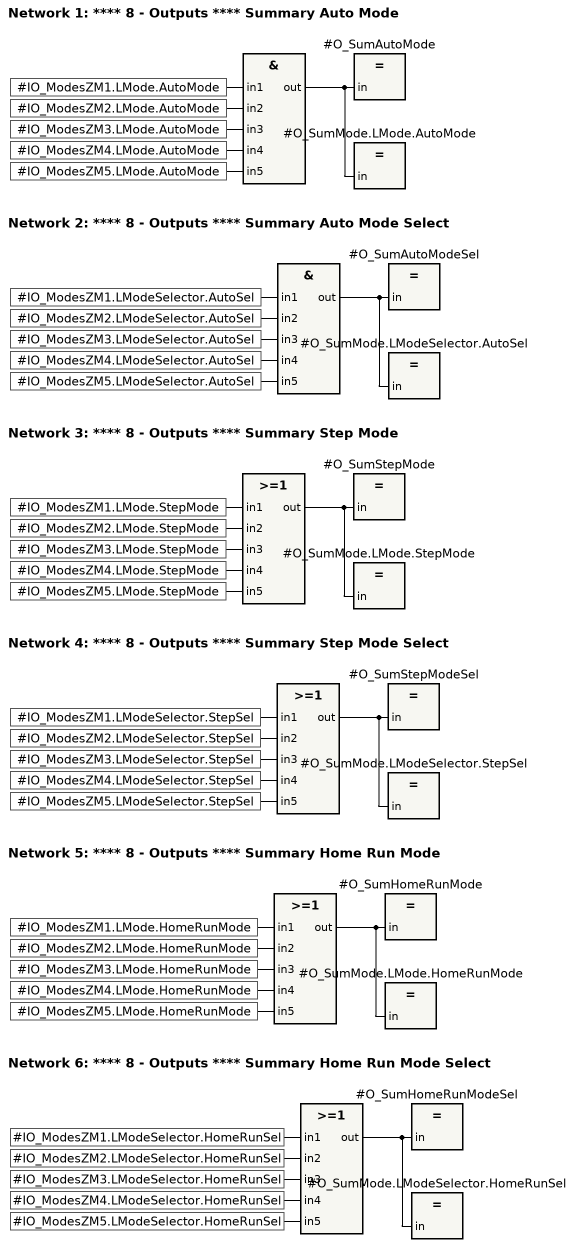
   #O_SumAutoMode := #IO_ModesZM1.LMode.AutoMode AND #IO_ModesZM2.LMode.AutoMode AND #IO_ModesZM3.LMode.AutoMode AND #IO_ModesZM4.LMode.AutoMode AND #IO_ModesZM5.LMode.AutoMode;
   #O_SumMode.LMode.AutoMode := #O_SumAutoMode;
END_REGION

REGION Network 2: **** 8 - Outputs **** Summary Auto Mode Select
   #O_SumAutoModeSel := #IO_ModesZM1.LModeSelector.AutoSel AND #IO_ModesZM2.LModeSelector.AutoSel AND #IO_ModesZM3.LModeSelector.AutoSel AND #IO_ModesZM4.LModeSelector.AutoSel AND #IO_ModesZM5.LModeSelector.AutoSel;
   #O_SumMode.LModeSelector.AutoSel := #O_SumAutoModeSel;
END_REGION

REGION Network 3: **** 8 - Outputs **** Summary Step Mode
   #O_SumStepMode := #IO_ModesZM1.LMode.StepMode OR #IO_ModesZM2.LMode.StepMode OR #IO_ModesZM3.LMode.StepMode OR #IO_ModesZM4.LMode.StepMode OR #IO_ModesZM5.LMode.StepMode;
   #O_SumMode.LMode.StepMode := #O_SumStepMode;
END_REGION

REGION Network 4: **** 8 - Outputs **** Summary Step Mode Select
   #O_SumStepModeSel := #IO_ModesZM1.LModeSelector.StepSel OR #IO_ModesZM2.LModeSelector.StepSel OR #IO_ModesZM3.LModeSelector.StepSel OR #IO_ModesZM4.LModeSelector.StepSel OR #IO_ModesZM5.LModeSelector.StepSel;
   #O_SumMode.LModeSelector.StepSel := #O_SumStepModeSel;
END_REGION

REGION Network 5: **** 8 - Outputs **** Summary Home Run Mode
   #O_SumHomeRunMode := #IO_ModesZM1.LMode.HomeRunMode OR #IO_ModesZM2.LMode.HomeRunMode OR #IO_ModesZM3.LMode.HomeRunMode OR #IO_ModesZM4.LMode.HomeRunMode OR #IO_ModesZM5.LMode.HomeRunMode;
   #O_SumMode.LMode.HomeRunMode := #O_SumHomeRunMode;
END_REGION

REGION Network 6: **** 8 - Outputs **** Summary Home Run Mode Select
   #O_SumHomeRunModeSel := #IO_ModesZM1.LModeSelector.HomeRunSel OR #IO_ModesZM2.LModeSelector.HomeRunSel OR #IO_ModesZM3.LModeSelector.HomeRunSel OR #IO_ModesZM4.LModeSelector.HomeRunSel OR #IO_ModesZM5.LModeSelector.HomeRunSel;
   #O_SumMode.LModeSelector.HomeRunSel := #O_SumHomeRunModeSel;
END_REGION

REGION Network 7: **** 8 - Outputs **** Summary Manual Mode
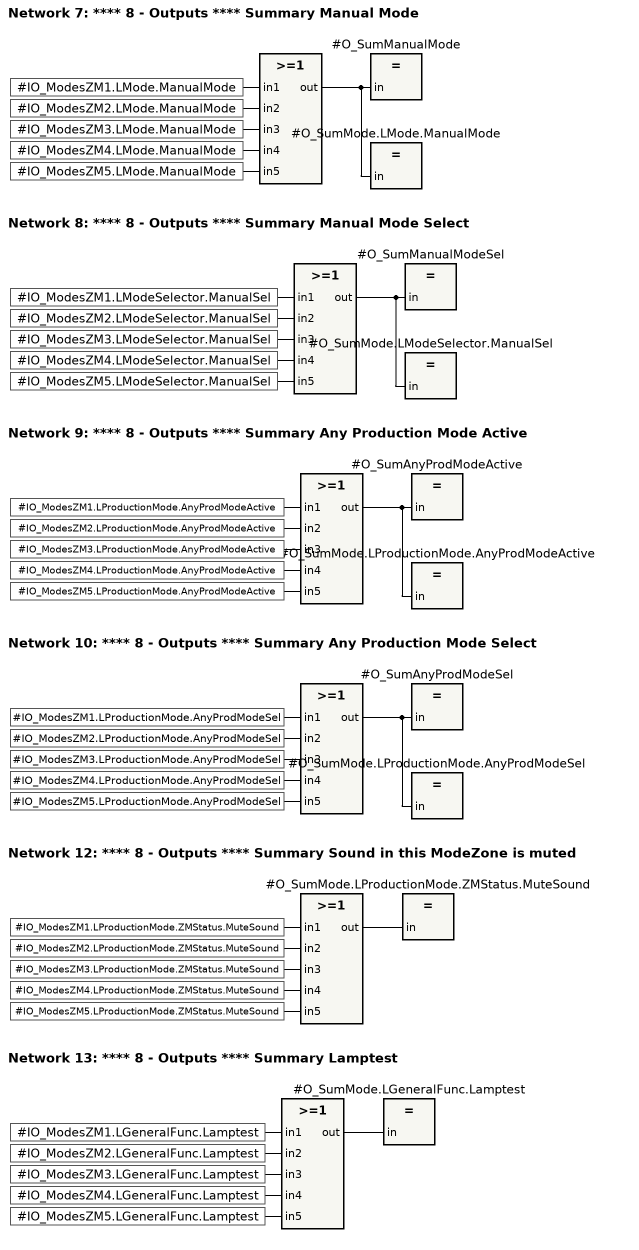
   #O_SumManualMode := #IO_ModesZM1.LMode.ManualMode OR #IO_ModesZM2.LMode.ManualMode OR #IO_ModesZM3.LMode.ManualMode OR #IO_ModesZM4.LMode.ManualMode OR #IO_ModesZM5.LMode.ManualMode;
   #O_SumMode.LMode.ManualMode := #O_SumManualMode;
END_REGION

REGION Network 8: **** 8 - Outputs **** Summary Manual Mode Select
   #O_SumManualModeSel := #IO_ModesZM1.LModeSelector.ManualSel OR #IO_ModesZM2.LModeSelector.ManualSel OR #IO_ModesZM3.LModeSelector.ManualSel OR #IO_ModesZM4.LModeSelector.ManualSel OR #IO_ModesZM5.LModeSelector.ManualSel;
   #O_SumMode.LModeSelector.ManualSel := #O_SumManualModeSel;
END_REGION

REGION Network 9: **** 8 - Outputs **** Summary Any Production Mode Active
   #O_SumAnyProdModeActive := #IO_ModesZM1.LProductionMode.AnyProdModeActive OR #IO_ModesZM2.LProductionMode.AnyProdModeActive OR #IO_ModesZM3.LProductionMode.AnyProdModeActive OR #IO_ModesZM4.LProductionMode.AnyProdModeActive OR #IO_ModesZM5.LProductionMode.AnyProdModeActive;
   #O_SumMode.LProductionMode.AnyProdModeActive := #O_SumAnyProdModeActive;
END_REGION

REGION Network 10: **** 8 - Outputs **** Summary Any Production Mode Select
   #O_SumAnyProdModeSel := #IO_ModesZM1.LProductionMode.AnyProdModeSel OR #IO_ModesZM2.LProductionMode.AnyProdModeSel OR #IO_ModesZM3.LProductionMode.AnyProdModeSel OR #IO_ModesZM4.LProductionMode.AnyProdModeSel OR #IO_ModesZM5.LProductionMode.AnyProdModeSel;
   #O_SumMode.LProductionMode.AnyProdModeSel := #O_SumAnyProdModeSel;
END_REGION

REGION Network 11: **** --------------------- Extra --------------------- ****
END_REGION

REGION Network 12: **** 8 - Outputs **** Summary Sound in this ModeZone is muted
   #O_SumMode.LProductionMode.ZMStatus.MuteSound := #IO_ModesZM1.LProductionMode.ZMStatus.MuteSound OR #IO_ModesZM2.LProductionMode.ZMStatus.MuteSound OR #IO_ModesZM3.LProductionMode.ZMStatus.MuteSound OR #IO_ModesZM4.LProductionMode.ZMStatus.MuteSound OR #IO_ModesZM5.LProductionMode.ZMStatus.MuteSound;
END_REGION

REGION Network 13: **** 8 - Outputs **** Summary Lamptest
   #O_SumMode.LGeneralFunc.Lamptest := #IO_ModesZM1.LGeneralFunc.Lamptest OR #IO_ModesZM2.LGeneralFunc.Lamptest OR #IO_ModesZM3.LGeneralFunc.Lamptest OR #IO_ModesZM4.LGeneralFunc.Lamptest OR #IO_ModesZM5.LGeneralFunc.Lamptest;
END_REGION

REGION Network 14: ***** 8 - Outputs **** Summary Lamptest steady
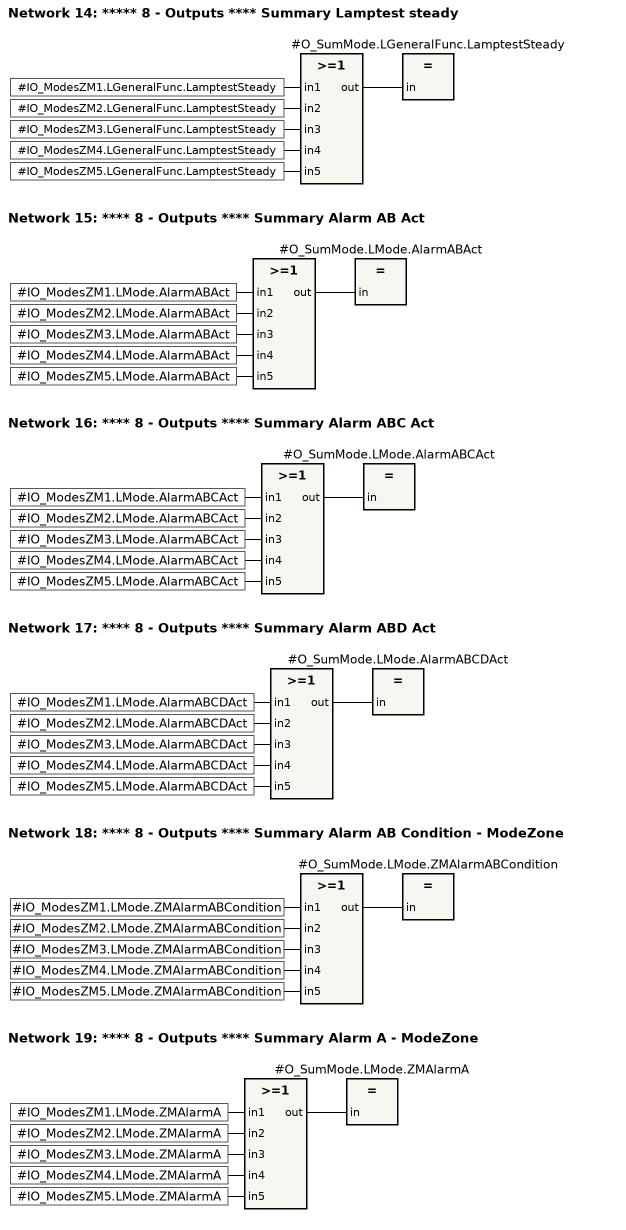
   #O_SumMode.LGeneralFunc.LamptestSteady := #IO_ModesZM1.LGeneralFunc.LamptestSteady OR #IO_ModesZM2.LGeneralFunc.LamptestSteady OR #IO_ModesZM3.LGeneralFunc.LamptestSteady OR #IO_ModesZM4.LGeneralFunc.LamptestSteady OR #IO_ModesZM5.LGeneralFunc.LamptestSteady;
END_REGION

REGION Network 15: **** 8 - Outputs **** Summary Alarm AB Act
   #O_SumMode.LMode.AlarmABAct := #IO_ModesZM1.LMode.AlarmABAct OR #IO_ModesZM2.LMode.AlarmABAct OR #IO_ModesZM3.LMode.AlarmABAct OR #IO_ModesZM4.LMode.AlarmABAct OR #IO_ModesZM5.LMode.AlarmABAct;
END_REGION

REGION Network 16: **** 8 - Outputs **** Summary Alarm ABC Act
   #O_SumMode.LMode.AlarmABCAct := #IO_ModesZM1.LMode.AlarmABCAct OR #IO_ModesZM2.LMode.AlarmABCAct OR #IO_ModesZM3.LMode.AlarmABCAct OR #IO_ModesZM4.LMode.AlarmABCAct OR #IO_ModesZM5.LMode.AlarmABCAct;
END_REGION

REGION Network 17: **** 8 - Outputs **** Summary Alarm ABD Act
   #O_SumMode.LMode.AlarmABCDAct := #IO_ModesZM1.LMode.AlarmABCDAct OR #IO_ModesZM2.LMode.AlarmABCDAct OR #IO_ModesZM3.LMode.AlarmABCDAct OR #IO_ModesZM4.LMode.AlarmABCDAct OR #IO_ModesZM5.LMode.AlarmABCDAct;
END_REGION

REGION Network 18: **** 8 - Outputs **** Summary Alarm AB Condition - ModeZone
   #O_SumMode.LMode.ZMAlarmABCondition := #IO_ModesZM1.LMode.ZMAlarmABCondition OR #IO_ModesZM2.LMode.ZMAlarmABCondition OR #IO_ModesZM3.LMode.ZMAlarmABCondition OR #IO_ModesZM4.LMode.ZMAlarmABCondition OR #IO_ModesZM5.LMode.ZMAlarmABCondition;
END_REGION

REGION Network 19: **** 8 - Outputs **** Summary Alarm A - ModeZone
   #O_SumMode.LMode.ZMAlarmA := #IO_ModesZM1.LMode.ZMAlarmA OR #IO_ModesZM2.LMode.ZMAlarmA OR #IO_ModesZM3.LMode.ZMAlarmA OR #IO_ModesZM4.LMode.ZMAlarmA OR #IO_ModesZM5.LMode.ZMAlarmA;
END_REGION

REGION Network 20: **** 8 - Outputs **** Summary Alarm B - ModeZone
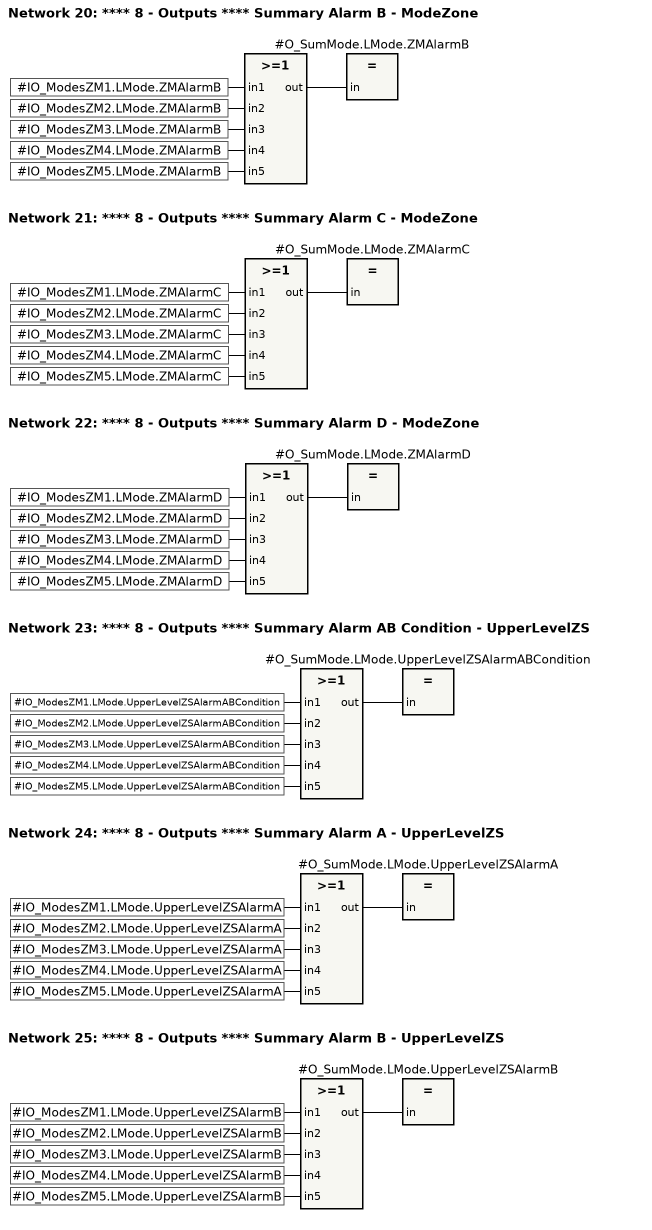
   #O_SumMode.LMode.ZMAlarmB := #IO_ModesZM1.LMode.ZMAlarmB OR #IO_ModesZM2.LMode.ZMAlarmB OR #IO_ModesZM3.LMode.ZMAlarmB OR #IO_ModesZM4.LMode.ZMAlarmB OR #IO_ModesZM5.LMode.ZMAlarmB;
END_REGION

REGION Network 21: **** 8 - Outputs **** Summary Alarm C - ModeZone
   #O_SumMode.LMode.ZMAlarmC := #IO_ModesZM1.LMode.ZMAlarmC OR #IO_ModesZM2.LMode.ZMAlarmC OR #IO_ModesZM3.LMode.ZMAlarmC OR #IO_ModesZM4.LMode.ZMAlarmC OR #IO_ModesZM5.LMode.ZMAlarmC;
END_REGION

REGION Network 22: **** 8 - Outputs **** Summary Alarm D - ModeZone
   #O_SumMode.LMode.ZMAlarmD := #IO_ModesZM1.LMode.ZMAlarmD OR #IO_ModesZM2.LMode.ZMAlarmD OR #IO_ModesZM3.LMode.ZMAlarmD OR #IO_ModesZM4.LMode.ZMAlarmD OR #IO_ModesZM5.LMode.ZMAlarmD;
END_REGION

REGION Network 23: **** 8 - Outputs **** Summary Alarm AB Condition - UpperLevelZS
   #O_SumMode.LMode.UpperLevelZSAlarmABCondition := #IO_ModesZM1.LMode.UpperLevelZSAlarmABCondition OR #IO_ModesZM2.LMode.UpperLevelZSAlarmABCondition OR #IO_ModesZM3.LMode.UpperLevelZSAlarmABCondition OR #IO_ModesZM4.LMode.UpperLevelZSAlarmABCondition OR #IO_ModesZM5.LMode.UpperLevelZSAlarmABCondition;
END_REGION

REGION Network 24: **** 8 - Outputs **** Summary Alarm A - UpperLevelZS
   #O_SumMode.LMode.UpperLevelZSAlarmA := #IO_ModesZM1.LMode.UpperLevelZSAlarmA OR #IO_ModesZM2.LMode.UpperLevelZSAlarmA OR #IO_ModesZM3.LMode.UpperLevelZSAlarmA OR #IO_ModesZM4.LMode.UpperLevelZSAlarmA OR #IO_ModesZM5.LMode.UpperLevelZSAlarmA;
END_REGION

REGION Network 25: **** 8 - Outputs **** Summary Alarm B - UpperLevelZS
   #O_SumMode.LMode.UpperLevelZSAlarmB := #IO_ModesZM1.LMode.UpperLevelZSAlarmB OR #IO_ModesZM2.LMode.UpperLevelZSAlarmB OR #IO_ModesZM3.LMode.UpperLevelZSAlarmB OR #IO_ModesZM4.LMode.UpperLevelZSAlarmB OR #IO_ModesZM5.LMode.UpperLevelZSAlarmB;
END_REGION

REGION Network 26: **** 8 - Outputs **** Summary Alarm C - UpperLevelZS
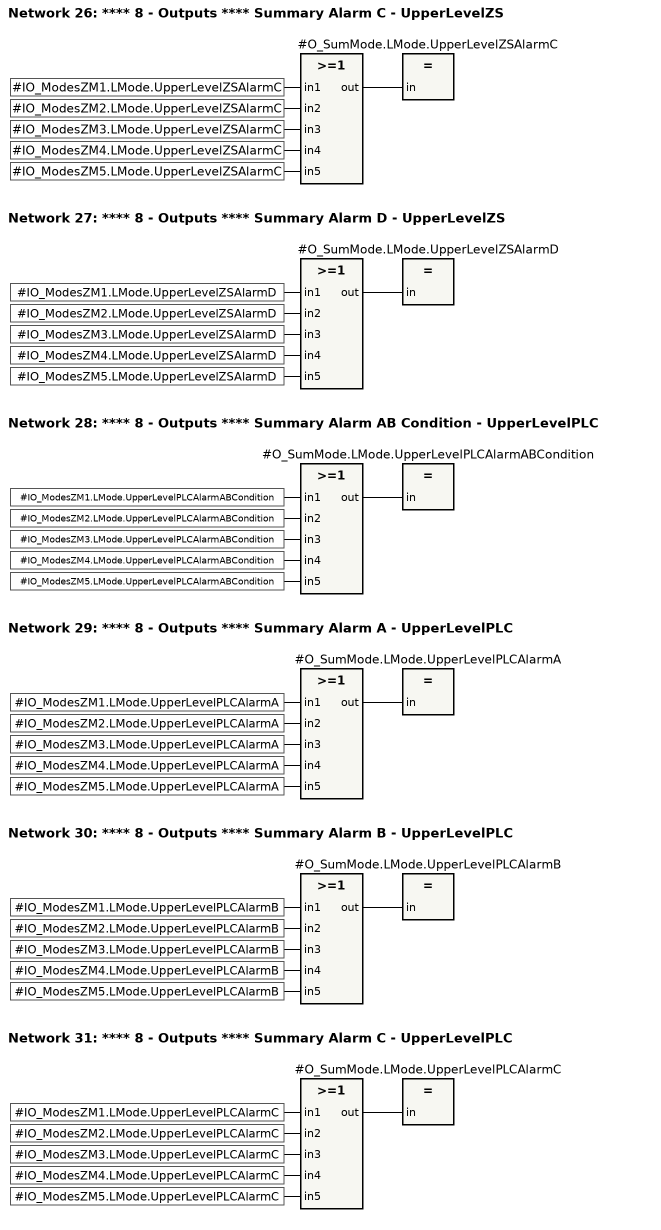
   #O_SumMode.LMode.UpperLevelZSAlarmC := #IO_ModesZM1.LMode.UpperLevelZSAlarmC OR #IO_ModesZM2.LMode.UpperLevelZSAlarmC OR #IO_ModesZM3.LMode.UpperLevelZSAlarmC OR #IO_ModesZM4.LMode.UpperLevelZSAlarmC OR #IO_ModesZM5.LMode.UpperLevelZSAlarmC;
END_REGION

REGION Network 27: **** 8 - Outputs **** Summary Alarm D - UpperLevelZS
   #O_SumMode.LMode.UpperLevelZSAlarmD := #IO_ModesZM1.LMode.UpperLevelZSAlarmD OR #IO_ModesZM2.LMode.UpperLevelZSAlarmD OR #IO_ModesZM3.LMode.UpperLevelZSAlarmD OR #IO_ModesZM4.LMode.UpperLevelZSAlarmD OR #IO_ModesZM5.LMode.UpperLevelZSAlarmD;
END_REGION

REGION Network 28: **** 8 - Outputs **** Summary Alarm AB Condition - UpperLevelPLC
   #O_SumMode.LMode.UpperLevelPLCAlarmABCondition := #IO_ModesZM1.LMode.UpperLevelPLCAlarmABCondition OR #IO_ModesZM2.LMode.UpperLevelPLCAlarmABCondition OR #IO_ModesZM3.LMode.UpperLevelPLCAlarmABCondition OR #IO_ModesZM4.LMode.UpperLevelPLCAlarmABCondition OR #IO_ModesZM5.LMode.UpperLevelPLCAlarmABCondition;
END_REGION

REGION Network 29: **** 8 - Outputs **** Summary Alarm A - UpperLevelPLC
   #O_SumMode.LMode.UpperLevelPLCAlarmA := #IO_ModesZM1.LMode.UpperLevelPLCAlarmA OR #IO_ModesZM2.LMode.UpperLevelPLCAlarmA OR #IO_ModesZM3.LMode.UpperLevelPLCAlarmA OR #IO_ModesZM4.LMode.UpperLevelPLCAlarmA OR #IO_ModesZM5.LMode.UpperLevelPLCAlarmA;
END_REGION

REGION Network 30: **** 8 - Outputs **** Summary Alarm B - UpperLevelPLC
   #O_SumMode.LMode.UpperLevelPLCAlarmB := #IO_ModesZM1.LMode.UpperLevelPLCAlarmB OR #IO_ModesZM2.LMode.UpperLevelPLCAlarmB OR #IO_ModesZM3.LMode.UpperLevelPLCAlarmB OR #IO_ModesZM4.LMode.UpperLevelPLCAlarmB OR #IO_ModesZM5.LMode.UpperLevelPLCAlarmB;
END_REGION

REGION Network 31: **** 8 - Outputs **** Summary Alarm C - UpperLevelPLC
   #O_SumMode.LMode.UpperLevelPLCAlarmC := #IO_ModesZM1.LMode.UpperLevelPLCAlarmC OR #IO_ModesZM2.LMode.UpperLevelPLCAlarmC OR #IO_ModesZM3.LMode.UpperLevelPLCAlarmC OR #IO_ModesZM4.LMode.UpperLevelPLCAlarmC OR #IO_ModesZM5.LMode.UpperLevelPLCAlarmC;
END_REGION

REGION Network 32: **** 8 - Outputs **** Summary Alarm D - UpperLevelPLC
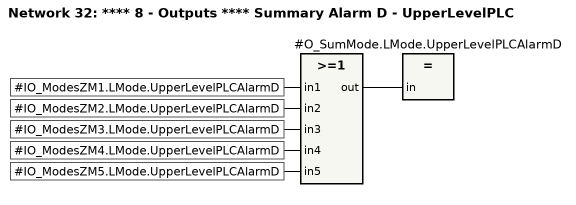
   #O_SumMode.LMode.UpperLevelPLCAlarmD := #IO_ModesZM1.LMode.UpperLevelPLCAlarmD OR #IO_ModesZM2.LMode.UpperLevelPLCAlarmD OR #IO_ModesZM3.LMode.UpperLevelPLCAlarmD OR #IO_ModesZM4.LMode.UpperLevelPLCAlarmD OR #IO_ModesZM5.LMode.UpperLevelPLCAlarmD;
END_REGION

REGION Network 33: **** -------------------------------------------------- ****
END_REGION
END_FUNCTION_BLOCK

FUNCTION_BLOCK "LModeSelectorHW"   // FB1005, FBD
TITLE = LModeSelectorHW
{ S7_Optimized_Access := 'FALSE' }
AUTHOR : VCC
FAMILY : Control
NAME : ModeSel
VERSION : 0.1
// ================================================================================
// This module handles that only one mode is selected in the modezon, it also 
// handle interlocking between the HMIs and panels. Each modezone can have 10 HMI.
// ================================================================================
// stored: AutoNumber false, IsIECCheckEnabled false, SetENOAutomatically False, UDAEnableTagReadback false
   VAR_INPUT
      I_NumHMI { ExternalAccessible := 'False'; ExternalVisible := 'False'; ExternalWritable := 'False'} : Int;   // Number of HMI used in the modezon
      I_StartPB { ExternalAccessible := 'False'; ExternalVisible := 'False'; ExternalWritable := 'False'} : Bool;   // Summary of Start buttons
      I_AlarmResetPB { ExternalAccessible := 'False'; ExternalVisible := 'False'; ExternalWritable := 'False'} : Bool;   // Summary of Alarm reset buttons
      I_HMI1ForceMan { ExternalAccessible := 'False'; ExternalVisible := 'False'; ExternalWritable := 'False'} : Bool;   // Forced manual selected on HMI1
      I_HMI1SetPB { ExternalAccessible := 'False'; ExternalVisible := 'False'; ExternalWritable := 'False'} : Bool;   // Set PB activated on HMI1
      I_HMI1ResetPB { ExternalAccessible := 'False'; ExternalVisible := 'False'; ExternalWritable := 'False'} : Bool;   // Reset PB activated on HMI1
      I_HMI1StartPB { ExternalAccessible := 'False'; ExternalVisible := 'False'; ExternalWritable := 'False'} : Bool;   // Start PB activated on HMI1
      I_HMI1AlarmResetPB { ExternalAccessible := 'False'; ExternalVisible := 'False'; ExternalWritable := 'False'} : Bool;   // AlarmReset PB activated on HMI1
      I_HMI1ResetSeqPB { ExternalAccessible := 'False'; ExternalVisible := 'False'; ExternalWritable := 'False'} : Bool;   // Reset Sequence PB
      I_HMI1ManSelSwitch { ExternalAccessible := 'False'; ExternalVisible := 'False'; ExternalWritable := 'False'} : Bool;   // Manual selection switch
      I_HMI1AutoSelSwitch { ExternalAccessible := 'False'; ExternalVisible := 'False'; ExternalWritable := 'False'} : Bool;   // Auto selection switch
      I_HMI2ForceMan { ExternalAccessible := 'False'; ExternalVisible := 'False'; ExternalWritable := 'False'} : Bool;   // Forced manual selected on HMI2
      I_HMI2SetPB { ExternalAccessible := 'False'; ExternalVisible := 'False'; ExternalWritable := 'False'} : Bool;   // Set PB activated on HMI2
      I_HMI2ResetPB { ExternalAccessible := 'False'; ExternalVisible := 'False'; ExternalWritable := 'False'} : Bool;   // Reset PB activated on HMI2
      I_HMI2StartPB { ExternalAccessible := 'False'; ExternalVisible := 'False'; ExternalWritable := 'False'} : Bool;   // Start PB activated on HMI2
      I_HMI2AlarmResetPB { ExternalAccessible := 'False'; ExternalVisible := 'False'; ExternalWritable := 'False'} : Bool;   // AlarmReset PB activated on HMI2
      I_HMI2ResetSeqPB { ExternalAccessible := 'False'; ExternalVisible := 'False'; ExternalWritable := 'False'} : Bool;   // Reset Sequence PB
      I_HMI2ManSelSwitch { ExternalAccessible := 'False'; ExternalVisible := 'False'; ExternalWritable := 'False'} : Bool;   // Manual selection switch
      I_HMI2AutoSelSwitch { ExternalAccessible := 'False'; ExternalVisible := 'False'; ExternalWritable := 'False'} : Bool;   // Auto selection switch
      I_HMI3ForceMan { ExternalAccessible := 'False'; ExternalVisible := 'False'; ExternalWritable := 'False'} : Bool;   // Forced manual selected on HMI3
      I_HMI3SetPB { ExternalAccessible := 'False'; ExternalVisible := 'False'; ExternalWritable := 'False'} : Bool;   // Set PB activated on HMI3
      I_HMI3ResetPB { ExternalAccessible := 'False'; ExternalVisible := 'False'; ExternalWritable := 'False'} : Bool;   // Reset PB activated on HMI3
      I_HMI3StartPB { ExternalAccessible := 'False'; ExternalVisible := 'False'; ExternalWritable := 'False'} : Bool;   // Start PB activated on HMI
      I_HMI3AlarmResetPB { ExternalAccessible := 'False'; ExternalVisible := 'False'; ExternalWritable := 'False'} : Bool;   // AlarmReset PB activated on HMI3
      I_HMI3ResetSeqPB { ExternalAccessible := 'False'; ExternalVisible := 'False'; ExternalWritable := 'False'} : Bool;   // Reset Sequence PB
      I_HMI3ManSelSwitch { ExternalAccessible := 'False'; ExternalVisible := 'False'; ExternalWritable := 'False'} : Bool;   // Manual selection switch
      I_HMI3AutoSelSwitch { ExternalAccessible := 'False'; ExternalVisible := 'False'; ExternalWritable := 'False'} : Bool;   // Auto selection switch
      I_HMI4ForceMan { ExternalAccessible := 'False'; ExternalVisible := 'False'; ExternalWritable := 'False'} : Bool;   // Forced manual selected on HMI4
      I_HMI4SetPB { ExternalAccessible := 'False'; ExternalVisible := 'False'; ExternalWritable := 'False'} : Bool;   // Set PB activated on HMI4
      I_HMI4ResetPB { ExternalAccessible := 'False'; ExternalVisible := 'False'; ExternalWritable := 'False'} : Bool;   // Reset PB activated on HMI4
      I_HMI4StartPB { ExternalAccessible := 'False'; ExternalVisible := 'False'; ExternalWritable := 'False'} : Bool;   // Start PB activated on HMI4
      I_HMI4AlarmResetPB { ExternalAccessible := 'False'; ExternalVisible := 'False'; ExternalWritable := 'False'} : Bool;   // AlarmReset PB activated on HMI4
      I_HMI4ResetSeqPB { ExternalAccessible := 'False'; ExternalVisible := 'False'; ExternalWritable := 'False'} : Bool;   // Reset Sequence PB
      I_HMI4ManSelSwitch { ExternalAccessible := 'False'; ExternalVisible := 'False'; ExternalWritable := 'False'} : Bool;   // Manual selection switch
      I_HMI4AutoSelSwitch { ExternalAccessible := 'False'; ExternalVisible := 'False'; ExternalWritable := 'False'} : Bool;   // Auto selection switch
      I_HMI5ForceMan { ExternalAccessible := 'False'; ExternalVisible := 'False'; ExternalWritable := 'False'} : Bool;   // Forced manual selected on HMI5
      I_HMI5SetPB { ExternalAccessible := 'False'; ExternalVisible := 'False'; ExternalWritable := 'False'} : Bool;   // Set PB activated on HMI5
      I_HMI5ResetPB { ExternalAccessible := 'False'; ExternalVisible := 'False'; ExternalWritable := 'False'} : Bool;   // Reset PB activated on HMI5
      I_HMI5StartPB { ExternalAccessible := 'False'; ExternalVisible := 'False'; ExternalWritable := 'False'} : Bool;   // Start PB activated on HMI5
      I_HMI5AlarmResetPB { ExternalAccessible := 'False'; ExternalVisible := 'False'; ExternalWritable := 'False'} : Bool;   // AlarmReset PB activated on HMI5
      I_HMI5ResetSeqPB { ExternalAccessible := 'False'; ExternalVisible := 'False'; ExternalWritable := 'False'} : Bool;   // Reset Sequence PB
      I_HMI5ManSelSwitch { ExternalAccessible := 'False'; ExternalVisible := 'False'; ExternalWritable := 'False'} : Bool;   // Manual selection switch
      I_HMI5AutoSelSwitch { ExternalAccessible := 'False'; ExternalVisible := 'False'; ExternalWritable := 'False'} : Bool;   // Auto selection switch
      I_HMI6ForceMan { ExternalAccessible := 'False'; ExternalVisible := 'False'; ExternalWritable := 'False'} : Bool;   // Forced manual selected on HMI6
      I_HMI6SetPB { ExternalAccessible := 'False'; ExternalVisible := 'False'; ExternalWritable := 'False'} : Bool;   // Set PB activated on HMI6
      I_HMI6ResetPB { ExternalAccessible := 'False'; ExternalVisible := 'False'; ExternalWritable := 'False'} : Bool;   // Reset PB activated on HMI6
      I_HMI6StartPB { ExternalAccessible := 'False'; ExternalVisible := 'False'; ExternalWritable := 'False'} : Bool;   // Start PB activated on HMI6
      I_HMI6AlarmResetPB { ExternalAccessible := 'False'; ExternalVisible := 'False'; ExternalWritable := 'False'} : Bool;   // AlarmReset PB activated on HMI6
      I_HMI6ResetSeqPB { ExternalAccessible := 'False'; ExternalVisible := 'False'; ExternalWritable := 'False'} : Bool;   // Reset Sequence PB
      I_HMI6ManSelSwitch { ExternalAccessible := 'False'; ExternalVisible := 'False'; ExternalWritable := 'False'} : Bool;   // Manual selection switch
      I_HMI6AutoSelSwitch { ExternalAccessible := 'False'; ExternalVisible := 'False'; ExternalWritable := 'False'} : Bool;   // Auto selection switch
      I_HMI7ForceMan { ExternalAccessible := 'False'; ExternalVisible := 'False'; ExternalWritable := 'False'} : Bool;   // Forced manual selected on HMI7
      I_HMI7SetPB { ExternalAccessible := 'False'; ExternalVisible := 'False'; ExternalWritable := 'False'} : Bool;   // Set PB activated on HMI7
      I_HMI7ResetPB { ExternalAccessible := 'False'; ExternalVisible := 'False'; ExternalWritable := 'False'} : Bool;   // Reset PB activated on HMI7
      I_HMI7StartPB { ExternalAccessible := 'False'; ExternalVisible := 'False'; ExternalWritable := 'False'} : Bool;   // Start PB activated on HMI7
      I_HMI7AlarmResetPB { ExternalAccessible := 'False'; ExternalVisible := 'False'; ExternalWritable := 'False'} : Bool;   // AlarmReset PB activated on HMI7
      I_HMI7ResetSeqPB { ExternalAccessible := 'False'; ExternalVisible := 'False'; ExternalWritable := 'False'} : Bool;   // Reset Sequence PB
      I_HMI7ManSelSwitch { ExternalAccessible := 'False'; ExternalVisible := 'False'; ExternalWritable := 'False'} : Bool;   // Manual selection switch
      I_HMI7AutoSelSwitch { ExternalAccessible := 'False'; ExternalVisible := 'False'; ExternalWritable := 'False'} : Bool;   // Auto selection switch
      I_HMI8ForceMan { ExternalAccessible := 'False'; ExternalVisible := 'False'; ExternalWritable := 'False'} : Bool;   // Forced manual selected on HMI8
      I_HMI8SetPB { ExternalAccessible := 'False'; ExternalVisible := 'False'; ExternalWritable := 'False'} : Bool;   // Set PB activated on HMI8
      I_HMI8ResetPB { ExternalAccessible := 'False'; ExternalVisible := 'False'; ExternalWritable := 'False'} : Bool;   // Reset PB activated on HMI8
      I_HMI8StartPB { ExternalAccessible := 'False'; ExternalVisible := 'False'; ExternalWritable := 'False'} : Bool;   // Start PB activated on HMI8
      I_HMI8AlarmResetPB { ExternalAccessible := 'False'; ExternalVisible := 'False'; ExternalWritable := 'False'} : Bool;   // AlarmReset PB activated on HMI8
      I_HMI8ResetSeqPB { ExternalAccessible := 'False'; ExternalVisible := 'False'; ExternalWritable := 'False'} : Bool;   // Reset Sequence PB
      I_HMI8ManSelSwitch { ExternalAccessible := 'False'; ExternalVisible := 'False'; ExternalWritable := 'False'} : Bool;   // Manual selection switch
      I_HMI8AutoSelSwitch { ExternalAccessible := 'False'; ExternalVisible := 'False'; ExternalWritable := 'False'} : Bool;   // Auto selection switch
      I_HMI9ForceMan { ExternalAccessible := 'False'; ExternalVisible := 'False'; ExternalWritable := 'False'} : Bool;   // Forced manual selected on HMI9
      I_HMI9SetPB { ExternalAccessible := 'False'; ExternalVisible := 'False'; ExternalWritable := 'False'} : Bool;   // Set PB activated on HMI9
      I_HMI9ResetPB { ExternalAccessible := 'False'; ExternalVisible := 'False'; ExternalWritable := 'False'} : Bool;   // Reset PB activated on HMI9
      I_HMI9StartPB { ExternalAccessible := 'False'; ExternalVisible := 'False'; ExternalWritable := 'False'} : Bool;   // Start PB activated on HMI9
      I_HMI9AlarmResetPB { ExternalAccessible := 'False'; ExternalVisible := 'False'; ExternalWritable := 'False'} : Bool;   // AlarmReset PB activated on HMI9
      I_HMI9ResetSeqPB { ExternalAccessible := 'False'; ExternalVisible := 'False'; ExternalWritable := 'False'} : Bool;   // Reset Sequence PB
      I_HMI9ManSelSwitch { ExternalAccessible := 'False'; ExternalVisible := 'False'; ExternalWritable := 'False'} : Bool;   // Manual selection switch
      I_HMI9AutoSelSwitch { ExternalAccessible := 'False'; ExternalVisible := 'False'; ExternalWritable := 'False'} : Bool;   // Auto selection switch
      I_HMI10ForceMan { ExternalAccessible := 'False'; ExternalVisible := 'False'; ExternalWritable := 'False'} : Bool;   // Forced manual selected on HMI10
      I_HMI10SetPB { ExternalAccessible := 'False'; ExternalVisible := 'False'; ExternalWritable := 'False'} : Bool;   // Set PB activated on HMI10
      I_HMI10ResetPB { ExternalAccessible := 'False'; ExternalVisible := 'False'; ExternalWritable := 'False'} : Bool;   // Reset PB activated on HMI10
      I_HMI10StartPB { ExternalAccessible := 'False'; ExternalVisible := 'False'; ExternalWritable := 'False'} : Bool;   // Start PB activated on HMI10
      I_HMI10AlarmResetPB { ExternalAccessible := 'False'; ExternalVisible := 'False'; ExternalWritable := 'False'} : Bool;   // AlarmReset PB activated on HMI10
      I_HMI10ResetSeqPB { ExternalAccessible := 'False'; ExternalVisible := 'False'; ExternalWritable := 'False'} : Bool;   // Reset Sequence PB
      I_HMI10ManSelSwitch { ExternalAccessible := 'False'; ExternalVisible := 'False'; ExternalWritable := 'False'} : Bool;   // Manual selection switch
      I_HMI10AutoSelSwitch { ExternalAccessible := 'False'; ExternalVisible := 'False'; ExternalWritable := 'False'} : Bool;   // Auto selection switch
      C_HMI1HW { ExternalAccessible := 'False'; ExternalVisible := 'False'; ExternalWritable := 'False'} : Bool;   // 1= HW OP panel. 0= Workstation
      C_HMI1SelectModes { ExternalAccessible := 'False'; ExternalVisible := 'False'; ExternalWritable := 'False'} : Bool;   // 1= This HMI can change the modes of this modezone
      C_HMI2HW { ExternalAccessible := 'False'; ExternalVisible := 'False'; ExternalWritable := 'False'} : Bool;   // 1= HW OP panel. 0= Workstation
      C_HMI2SelectModes { ExternalAccessible := 'False'; ExternalVisible := 'False'; ExternalWritable := 'False'} : Bool;   // 1= This HMI can change the modes of this modezone
      C_HMI3HW { ExternalAccessible := 'False'; ExternalVisible := 'False'; ExternalWritable := 'False'} : Bool;   // 1= HW OP panel. 0= Workstation
      C_HMI3SelectModes { ExternalAccessible := 'False'; ExternalVisible := 'False'; ExternalWritable := 'False'} : Bool;   // 1= This HMI can change the modes of this modezone
      C_HMI4HW { ExternalAccessible := 'False'; ExternalVisible := 'False'; ExternalWritable := 'False'} : Bool;   // 1= HW OP panel. 0= Workstation
      C_HMI4SelectModes { ExternalAccessible := 'False'; ExternalVisible := 'False'; ExternalWritable := 'False'} : Bool;   // 1= This HMI can change the modes of this modezone
      C_HMI5HW { ExternalAccessible := 'False'; ExternalVisible := 'False'; ExternalWritable := 'False'} : Bool;   // 1= HW OP panel. 0= Workstation
      C_HMI5SelectModes { ExternalAccessible := 'False'; ExternalVisible := 'False'; ExternalWritable := 'False'} : Bool;   // 1= This HMI can change the modes of this modezone
      C_HMI6HW { ExternalAccessible := 'False'; ExternalVisible := 'False'; ExternalWritable := 'False'} : Bool;   // 1= HW OP panel. 0= Workstation
      C_HMI6SelectModes { ExternalAccessible := 'False'; ExternalVisible := 'False'; ExternalWritable := 'False'} : Bool;   // 1= This HMI can change the modes of this modezone
      C_HMI7HW { ExternalAccessible := 'False'; ExternalVisible := 'False'; ExternalWritable := 'False'} : Bool;   // 1= HW OP panel. 0= Workstation
      C_HMI7SelectModes { ExternalAccessible := 'False'; ExternalVisible := 'False'; ExternalWritable := 'False'} : Bool;   // 1= This HMI can change the modes of this modezone
      C_HMI8HW { ExternalAccessible := 'False'; ExternalVisible := 'False'; ExternalWritable := 'False'} : Bool;   // 1= HW OP panel. 0= Workstation
      C_HMI8SelectModes { ExternalAccessible := 'False'; ExternalVisible := 'False'; ExternalWritable := 'False'} : Bool;   // 1= This HMI can change the modes of this modezone
      C_HMI9HW { ExternalAccessible := 'False'; ExternalVisible := 'False'; ExternalWritable := 'False'} : Bool;   // 1= HW OP panel. 0= Workstation
      C_HMI9SelectModes { ExternalAccessible := 'False'; ExternalVisible := 'False'; ExternalWritable := 'False'} : Bool;   // 1= This HMI can change the modes of this modezone
      C_HMI10HW { ExternalAccessible := 'False'; ExternalVisible := 'False'; ExternalWritable := 'False'} : Bool;   // 1= HW OP panel. 0= Workstation
      C_HMI10SelectModes { ExternalAccessible := 'False'; ExternalVisible := 'False'; ExternalWritable := 'False'} : Bool;   // 1= This HMI can change the modes of this modezone
   END_VAR
   VAR_OUTPUT
      O_ActiveHMI { ExternalAccessible := 'False'; ExternalVisible := 'False'; ExternalWritable := 'False'} : Int;   // Active HMI
      O_AutoSel { ExternalAccessible := 'False'; ExternalVisible := 'False'; ExternalWritable := 'False'} : Bool;   // Auto selected
      O_AllAutoSel { ExternalAccessible := 'False'; ExternalVisible := 'False'; ExternalWritable := 'False'} : Bool;   // All objects in Auto selected
      O_StepSel { ExternalAccessible := 'False'; ExternalVisible := 'False'; ExternalWritable := 'False'} : Bool;   // Step selected
      O_HomeRunSel { ExternalAccessible := 'False'; ExternalVisible := 'False'; ExternalWritable := 'False'} : Bool;   // Homerun selected
      O_ManualSel { ExternalAccessible := 'False'; ExternalVisible := 'False'; ExternalWritable := 'False'} : Bool;   // Manual selected
      O_ForcedManActSel { ExternalAccessible := 'False'; ExternalVisible := 'False'; ExternalWritable := 'False'} : Bool;   // Forced manual selected
      O_PBSetSel { ExternalAccessible := 'False'; ExternalVisible := 'False'; ExternalWritable := 'False'} : Bool;   // Set selected
      O_PBResetSel { ExternalAccessible := 'False'; ExternalVisible := 'False'; ExternalWritable := 'False'} : Bool;   // Reset selected
      O_StartPBSel { ExternalAccessible := 'False'; ExternalVisible := 'False'; ExternalWritable := 'False'} : Bool;   // Start is activated
      O_AlarmResetPBSel { ExternalAccessible := 'False'; ExternalVisible := 'False'; ExternalWritable := 'False'} : Bool;   // Alarm reset is activated
      O_ResetTMSel { ExternalAccessible := 'False'; ExternalVisible := 'False'; ExternalWritable := 'False'} : Bool;   // Reset transport memory
      O_ResetSeqSel { ExternalAccessible := 'False'; ExternalVisible := 'False'; ExternalWritable := 'False'} : Bool;   // Reset squence
      O_CycleFinishedSel { ExternalAccessible := 'False'; ExternalVisible := 'False'; ExternalWritable := 'False'} : Bool;   // Cycle finished selected
      O_HomeRunRedoSel { ExternalAccessible := 'False'; ExternalVisible := 'False'; ExternalWritable := 'False'} : Bool;   // Redo after Homerun selected
      O_HomeRunWorkDoneSel { ExternalAccessible := 'False'; ExternalVisible := 'False'; ExternalWritable := 'False'} : Bool;   // WorkDone after Homerun selected
   END_VAR
   VAR_IN_OUT
      IO_Modes : "Modes";
   END_VAR
   VAR DB_SPECIFIC
      H_HMIHomeRunModeCmd : Word;   // Homerun Mode commands from HMI
      H_Anim : Word;   // Animation for HMI
      H_ActiveHMI : Int;   // Active HMI
      H_NameActiveHMI : String[25];   // Name of the Active HMI
      H_LockManTime : Int;   // Lock manual time
      H_HMI1ModeCmd : Word;   // Mode commands from HMI1
      H_HMI2ModeCmd : Word;   // Mode commands from HMI2
      H_HMI3ModeCmd : Word;   // Mode commands from HMI3
      H_HMI4ModeCmd : Word;   // Mode commands from HMI4
      H_HMI5ModeCmd : Word;   // Mode commands from HMI5
      H_HMI6ModeCmd : Word;   // Mode commands from HMI6
      H_HMI7ModeCmd : Word;   // Mode commands from HMI7
      H_HMI8ModeCmd : Word;   // Mode commands from HMI8
      H_HMI9ModeCmd : Word;   // Mode commands from HMI9
      H_HMI10ModeCmd : Word;   // Mode commands from HMI10
      HMI1AutoSel { ExternalAccessible := 'False'; ExternalVisible := 'False'; ExternalWritable := 'False'} : Bool;   // Auto selected on HMI1
      HMI1StepSel { ExternalAccessible := 'False'; ExternalVisible := 'False'; ExternalWritable := 'False'} : Bool;   // Step selected on HMI1
      HMI1HomeRunSel { ExternalAccessible := 'False'; ExternalVisible := 'False'; ExternalWritable := 'False'} : Bool;   // Homerun selected on HMI1
      HMI1ManualSel { ExternalAccessible := 'False'; ExternalVisible := 'False'; ExternalWritable := 'False'} : Bool;   // Manual selected on HMI1
      HMI1LockManual { ExternalAccessible := 'False'; ExternalVisible := 'False'; ExternalWritable := 'False'} : Bool;   // Lock manual for HMI1
      HMI1AllHMIAutoSel { ExternalAccessible := 'False'; ExternalVisible := 'False'; ExternalWritable := 'False'} : Bool;   // All HMI Auto selected on HMI1
      HMI1Start { ExternalAccessible := 'False'; ExternalVisible := 'False'; ExternalWritable := 'False'} : Bool;   // Start on HMI1
      HMI1AlarmReset { ExternalAccessible := 'False'; ExternalVisible := 'False'; ExternalWritable := 'False'} : Bool;   // AlarmReset on HMI1
      HMI1ResetTM { ExternalAccessible := 'False'; ExternalVisible := 'False'; ExternalWritable := 'False'} : Bool;   // Reset transport memory from HMI1
      HMI1ResetSeq { ExternalAccessible := 'False'; ExternalVisible := 'False'; ExternalWritable := 'False'} : Bool;   // Reset sequence from HMI1
      HMI1CycleFinished { ExternalAccessible := 'False'; ExternalVisible := 'False'; ExternalWritable := 'False'} : Bool;   // Cycle Finished from HMI1
      HMI1AlarmResetAck { ExternalAccessible := 'False'; ExternalVisible := 'False'; ExternalWritable := 'False'} : Bool;   // Alarm Reset acknowledge from HMI1
      HMI2AutoSel { ExternalAccessible := 'False'; ExternalVisible := 'False'; ExternalWritable := 'False'} : Bool;   // Auto selected on HMI2
      HMI2StepSel { ExternalAccessible := 'False'; ExternalVisible := 'False'; ExternalWritable := 'False'} : Bool;   // Step selected on HMI2
      HMI2HomeRunSel { ExternalAccessible := 'False'; ExternalVisible := 'False'; ExternalWritable := 'False'} : Bool;   // Homerun selected on HMI2
      HMI2ManualSel { ExternalAccessible := 'False'; ExternalVisible := 'False'; ExternalWritable := 'False'} : Bool;   // Manual selected on HMI2
      HMI2LockManual { ExternalAccessible := 'False'; ExternalVisible := 'False'; ExternalWritable := 'False'} : Bool;   // Lock manual for HMI2
      HMI2AllHMIAutoSel { ExternalAccessible := 'False'; ExternalVisible := 'False'; ExternalWritable := 'False'} : Bool;   // All HMI Auto selected on HMI2
      HMI2Start { ExternalAccessible := 'False'; ExternalVisible := 'False'; ExternalWritable := 'False'} : Bool;   // Start on HMI2
      HMI2AlarmReset { ExternalAccessible := 'False'; ExternalVisible := 'False'; ExternalWritable := 'False'} : Bool;   // AlarmReset on HMI2
      HMI2ResetTM { ExternalAccessible := 'False'; ExternalVisible := 'False'; ExternalWritable := 'False'} : Bool;   // Reset transport memory from HMI2
      HMI2ResetSeq { ExternalAccessible := 'False'; ExternalVisible := 'False'; ExternalWritable := 'False'} : Bool;   // Reset sequence from HMI2
      HMI2CycleFinished { ExternalAccessible := 'False'; ExternalVisible := 'False'; ExternalWritable := 'False'} : Bool;   // Cycle Finished from HMI2
      HMI2AlarmResetAck { ExternalAccessible := 'False'; ExternalVisible := 'False'; ExternalWritable := 'False'} : Bool;   // Alarm Reset acknowledge from HMI2
      HMI3AutoSel { ExternalAccessible := 'False'; ExternalVisible := 'False'; ExternalWritable := 'False'} : Bool;   // Auto selected on HMI3
      HMI3StepSel { ExternalAccessible := 'False'; ExternalVisible := 'False'; ExternalWritable := 'False'} : Bool;   // Step selected on HMI3
      HMI3HomeRunSel { ExternalAccessible := 'False'; ExternalVisible := 'False'; ExternalWritable := 'False'} : Bool;   // Homerun selected on HMI3
      HMI3ManualSel { ExternalAccessible := 'False'; ExternalVisible := 'False'; ExternalWritable := 'False'} : Bool;   // Manual selected on HMI3
      HMI3LockManual { ExternalAccessible := 'False'; ExternalVisible := 'False'; ExternalWritable := 'False'} : Bool;   // Lock manual for HMI3
      HMI3AllHMIAutoSel { ExternalAccessible := 'False'; ExternalVisible := 'False'; ExternalWritable := 'False'} : Bool;   // All HMI Auto selected on HMI3
      HMI3Start { ExternalAccessible := 'False'; ExternalVisible := 'False'; ExternalWritable := 'False'} : Bool;   // Start on HMI3
      HMI3AlarmReset { ExternalAccessible := 'False'; ExternalVisible := 'False'; ExternalWritable := 'False'} : Bool;   // AlarmReset on HMI3
      HMI3ResetTM { ExternalAccessible := 'False'; ExternalVisible := 'False'; ExternalWritable := 'False'} : Bool;   // Reset transport memory from HMI3
      HMI3ResetSeq { ExternalAccessible := 'False'; ExternalVisible := 'False'; ExternalWritable := 'False'} : Bool;   // Reset sequence from HMI3
      HMI3CycleFinished { ExternalAccessible := 'False'; ExternalVisible := 'False'; ExternalWritable := 'False'} : Bool;   // Cycle Finished from HMI3
      HMI3AlarmResetAck { ExternalAccessible := 'False'; ExternalVisible := 'False'; ExternalWritable := 'False'} : Bool;   // Alarm Reset acknowledge from 3
      HMI4AutoSel { ExternalAccessible := 'False'; ExternalVisible := 'False'; ExternalWritable := 'False'} : Bool;   // Auto selected on HMI4
      HMI4StepSel { ExternalAccessible := 'False'; ExternalVisible := 'False'; ExternalWritable := 'False'} : Bool;   // Step selected on HMI4
      HMI4HomeRunSel { ExternalAccessible := 'False'; ExternalVisible := 'False'; ExternalWritable := 'False'} : Bool;   // Homerun selected on HMI4
      HMI4ManualSel { ExternalAccessible := 'False'; ExternalVisible := 'False'; ExternalWritable := 'False'} : Bool;   // Manual selected on HMI4
      HMI4LockManual { ExternalAccessible := 'False'; ExternalVisible := 'False'; ExternalWritable := 'False'} : Bool;   // Lock manual for HMI4
      HMI4AllHMIAutoSel { ExternalAccessible := 'False'; ExternalVisible := 'False'; ExternalWritable := 'False'} : Bool;   // All HMI Auto selected on HMI4
      HMI4Start { ExternalAccessible := 'False'; ExternalVisible := 'False'; ExternalWritable := 'False'} : Bool;   // Start on HMI4
      HMI4AlarmReset { ExternalAccessible := 'False'; ExternalVisible := 'False'; ExternalWritable := 'False'} : Bool;   // AlarmReset on HMI4
      HMI4ResetTM { ExternalAccessible := 'False'; ExternalVisible := 'False'; ExternalWritable := 'False'} : Bool;   // Reset transport memory from HMI4
      HMI4ResetSeq { ExternalAccessible := 'False'; ExternalVisible := 'False'; ExternalWritable := 'False'} : Bool;   // Reset sequence from HMI4
      HMI4CycleFinished { ExternalAccessible := 'False'; ExternalVisible := 'False'; ExternalWritable := 'False'} : Bool;   // Cycle Finished from HMI4
      HMI4AlarmResetAck { ExternalAccessible := 'False'; ExternalVisible := 'False'; ExternalWritable := 'False'} : Bool;   // Alarm Reset acknowledge from HMI4
      HMI5AutoSel { ExternalAccessible := 'False'; ExternalVisible := 'False'; ExternalWritable := 'False'} : Bool;   // Auto selected on HMI5
      HMI5StepSel { ExternalAccessible := 'False'; ExternalVisible := 'False'; ExternalWritable := 'False'} : Bool;   // Step selected on HMI5
      HMI5HomeRunSel { ExternalAccessible := 'False'; ExternalVisible := 'False'; ExternalWritable := 'False'} : Bool;   // Homerun selected on HMI5
      HMI5ManualSel { ExternalAccessible := 'False'; ExternalVisible := 'False'; ExternalWritable := 'False'} : Bool;   // Manual selected on HMI5
      HMI5LockManual { ExternalAccessible := 'False'; ExternalVisible := 'False'; ExternalWritable := 'False'} : Bool;   // Lock manual for HMI5
      HMI5AllHMIAutoSel { ExternalAccessible := 'False'; ExternalVisible := 'False'; ExternalWritable := 'False'} : Bool;   // All HMI Auto selected on HMI5
      HMI5Start { ExternalAccessible := 'False'; ExternalVisible := 'False'; ExternalWritable := 'False'} : Bool;   // Start on HMI5
      HMI5AlarmReset { ExternalAccessible := 'False'; ExternalVisible := 'False'; ExternalWritable := 'False'} : Bool;   // AlarmReset on HMI5
      HMI5ResetTM { ExternalAccessible := 'False'; ExternalVisible := 'False'; ExternalWritable := 'False'} : Bool;   // Reset transport memory from HMI5
      HMI5ResetSeq { ExternalAccessible := 'False'; ExternalVisible := 'False'; ExternalWritable := 'False'} : Bool;   // Reset sequence from HMI5
      HMI5CycleFinished { ExternalAccessible := 'False'; ExternalVisible := 'False'; ExternalWritable := 'False'} : Bool;   // Cycle Finished from HMI5
      HMI5AlarmResetAck { ExternalAccessible := 'False'; ExternalVisible := 'False'; ExternalWritable := 'False'} : Bool;   // Alarm Reset acknowledge from HMI5
      HMI6AutoSel { ExternalAccessible := 'False'; ExternalVisible := 'False'; ExternalWritable := 'False'} : Bool;   // Auto selected on HMI6
      HMI6StepSel { ExternalAccessible := 'False'; ExternalVisible := 'False'; ExternalWritable := 'False'} : Bool;   // Step selected on HMI6
      HMI6HomeRunSel { ExternalAccessible := 'False'; ExternalVisible := 'False'; ExternalWritable := 'False'} : Bool;   // Homerun selected on HMI6
      HMI6ManualSel { ExternalAccessible := 'False'; ExternalVisible := 'False'; ExternalWritable := 'False'} : Bool;   // Manual selected on HMI6
      HMI6LockManual { ExternalAccessible := 'False'; ExternalVisible := 'False'; ExternalWritable := 'False'} : Bool;   // Lock manual for HMI6
      HMI6AllHMIAutoSel { ExternalAccessible := 'False'; ExternalVisible := 'False'; ExternalWritable := 'False'} : Bool;   // All HMI Auto selected on HMI6
      HMI6Start { ExternalAccessible := 'False'; ExternalVisible := 'False'; ExternalWritable := 'False'} : Bool;   // Start on HMI6
      HMI6AlarmReset { ExternalAccessible := 'False'; ExternalVisible := 'False'; ExternalWritable := 'False'} : Bool;   // AlarmReset on HMI6
      HMI6ResetTM { ExternalAccessible := 'False'; ExternalVisible := 'False'; ExternalWritable := 'False'} : Bool;   // Reset transport memory from HMI6
      HMI6ResetSeq { ExternalAccessible := 'False'; ExternalVisible := 'False'; ExternalWritable := 'False'} : Bool;   // Reset sequence from HMI6
      HMI6CycleFinished { ExternalAccessible := 'False'; ExternalVisible := 'False'; ExternalWritable := 'False'} : Bool;   // Cycle Finished from HMI6
      HMI6AlarmResetAck { ExternalAccessible := 'False'; ExternalVisible := 'False'; ExternalWritable := 'False'} : Bool;   // Alarm Reset acknowledge from HMI6
      HMI7AutoSel { ExternalAccessible := 'False'; ExternalVisible := 'False'; ExternalWritable := 'False'} : Bool;   // Auto selected on HMI7
      HMI7StepSel { ExternalAccessible := 'False'; ExternalVisible := 'False'; ExternalWritable := 'False'} : Bool;   // Step selected on HMI7
      HMI7HomeRunSel { ExternalAccessible := 'False'; ExternalVisible := 'False'; ExternalWritable := 'False'} : Bool;   // Homerun selected on HMI7
      HMI7ManualSel { ExternalAccessible := 'False'; ExternalVisible := 'False'; ExternalWritable := 'False'} : Bool;   // Manual selected on HMI7
      HMI7LockManual { ExternalAccessible := 'False'; ExternalVisible := 'False'; ExternalWritable := 'False'} : Bool;   // Lock manual for HMI7
      HMI7AllHMIAutoSel { ExternalAccessible := 'False'; ExternalVisible := 'False'; ExternalWritable := 'False'} : Bool;   // All HMI Auto selected on HMI7
      HMI7Start { ExternalAccessible := 'False'; ExternalVisible := 'False'; ExternalWritable := 'False'} : Bool;   // Start on HMI7
      HMI7AlarmReset { ExternalAccessible := 'False'; ExternalVisible := 'False'; ExternalWritable := 'False'} : Bool;   // AlarmReset on HMI7
      HMI7ResetTM { ExternalAccessible := 'False'; ExternalVisible := 'False'; ExternalWritable := 'False'} : Bool;   // Reset transport memory from HMI7
      HMI7ResetSeq { ExternalAccessible := 'False'; ExternalVisible := 'False'; ExternalWritable := 'False'} : Bool;   // Reset sequence from HMI7
      HMI7CycleFinished { ExternalAccessible := 'False'; ExternalVisible := 'False'; ExternalWritable := 'False'} : Bool;   // Cycle Finished from HMI7
      HMI7AlarmResetAck { ExternalAccessible := 'False'; ExternalVisible := 'False'; ExternalWritable := 'False'} : Bool;   // Alarm Reset acknowledge from HMI7
      HMI8AutoSel { ExternalAccessible := 'False'; ExternalVisible := 'False'; ExternalWritable := 'False'} : Bool;   // Auto selected on HMI8
      HMI8StepSel { ExternalAccessible := 'False'; ExternalVisible := 'False'; ExternalWritable := 'False'} : Bool;   // Step selected on HMI8
      HMI8HomeRunSel { ExternalAccessible := 'False'; ExternalVisible := 'False'; ExternalWritable := 'False'} : Bool;   // Homerun selected on HMI8
      HMI8ManualSel { ExternalAccessible := 'False'; ExternalVisible := 'False'; ExternalWritable := 'False'} : Bool;   // Manual selected on HMI8
      HMI8LockManual { ExternalAccessible := 'False'; ExternalVisible := 'False'; ExternalWritable := 'False'} : Bool;   // Lock manual for HMI8
      HMI8AllHMIAutoSel { ExternalAccessible := 'False'; ExternalVisible := 'False'; ExternalWritable := 'False'} : Bool;   // All HMI Auto selected on HMI8
      HMI8Start { ExternalAccessible := 'False'; ExternalVisible := 'False'; ExternalWritable := 'False'} : Bool;   // Start on HMI8
      HMI8AlarmReset { ExternalAccessible := 'False'; ExternalVisible := 'False'; ExternalWritable := 'False'} : Bool;   // AlarmReset on HMI8
      HMI8ResetTM { ExternalAccessible := 'False'; ExternalVisible := 'False'; ExternalWritable := 'False'} : Bool;   // Reset transport memory from HMI8
      HMI8ResetSeq { ExternalAccessible := 'False'; ExternalVisible := 'False'; ExternalWritable := 'False'} : Bool;   // Reset sequence from HMI8
      HMI8CycleFinished { ExternalAccessible := 'False'; ExternalVisible := 'False'; ExternalWritable := 'False'} : Bool;   // Cycle Finished from HMI8
      HMI8AlarmResetAck { ExternalAccessible := 'False'; ExternalVisible := 'False'; ExternalWritable := 'False'} : Bool;   // Alarm Reset acknowledge from HMI8
      HMI9AutoSel { ExternalAccessible := 'False'; ExternalVisible := 'False'; ExternalWritable := 'False'} : Bool;   // Auto selected on HMI9
      HMI9StepSel { ExternalAccessible := 'False'; ExternalVisible := 'False'; ExternalWritable := 'False'} : Bool;   // Step selected on HMI9
      HMI9HomeRunSel { ExternalAccessible := 'False'; ExternalVisible := 'False'; ExternalWritable := 'False'} : Bool;   // Homerun selected on HMI9
      HMI9ManualSel { ExternalAccessible := 'False'; ExternalVisible := 'False'; ExternalWritable := 'False'} : Bool;   // Manual selected on HMI9
      HMI9LockManual { ExternalAccessible := 'False'; ExternalVisible := 'False'; ExternalWritable := 'False'} : Bool;   // Lock manual for HMI9
      HMI9AllHMIAutoSel { ExternalAccessible := 'False'; ExternalVisible := 'False'; ExternalWritable := 'False'} : Bool;   // All HMI Auto selected on HMI9
      HMI9Start { ExternalAccessible := 'False'; ExternalVisible := 'False'; ExternalWritable := 'False'} : Bool;   // Start on HMI9
      HMI9AlarmReset { ExternalAccessible := 'False'; ExternalVisible := 'False'; ExternalWritable := 'False'} : Bool;   // AlarmReset on HMI9
      HMI9ResetTM { ExternalAccessible := 'False'; ExternalVisible := 'False'; ExternalWritable := 'False'} : Bool;   // Reset transport memory from HMI9
      HMI9ResetSeq { ExternalAccessible := 'False'; ExternalVisible := 'False'; ExternalWritable := 'False'} : Bool;   // Reset sequence from HMI9
      HMI9CycleFinished { ExternalAccessible := 'False'; ExternalVisible := 'False'; ExternalWritable := 'False'} : Bool;   // Cycle Finished from HMI9
      HMI9AlarmResetAck { ExternalAccessible := 'False'; ExternalVisible := 'False'; ExternalWritable := 'False'} : Bool;   // Alarm Reset acknowledge from HMI9
      HMI10AutoSel { ExternalAccessible := 'False'; ExternalVisible := 'False'; ExternalWritable := 'False'} : Bool;   // Auto selected on HMI10
      HMI10StepSel { ExternalAccessible := 'False'; ExternalVisible := 'False'; ExternalWritable := 'False'} : Bool;   // Step selected on HMI10
      HMI10HomeRunSel { ExternalAccessible := 'False'; ExternalVisible := 'False'; ExternalWritable := 'False'} : Bool;   // Homerun selected on HMI10
      HMI10ManualSel { ExternalAccessible := 'False'; ExternalVisible := 'False'; ExternalWritable := 'False'} : Bool;   // Manual selected on HMI10
      HMI10LockManual { ExternalAccessible := 'False'; ExternalVisible := 'False'; ExternalWritable := 'False'} : Bool;   // Lock manual for HMI10
      HMI10AllHMIAutoSel { ExternalAccessible := 'False'; ExternalVisible := 'False'; ExternalWritable := 'False'} : Bool;   // All HMI Auto selected on HMI10
      HMI10Start { ExternalAccessible := 'False'; ExternalVisible := 'False'; ExternalWritable := 'False'} : Bool;   // Start on HMI10
      HMI10AlarmReset { ExternalAccessible := 'False'; ExternalVisible := 'False'; ExternalWritable := 'False'} : Bool;   // AlarmReset on HMI10
      HMI10ResetTM { ExternalAccessible := 'False'; ExternalVisible := 'False'; ExternalWritable := 'False'} : Bool;   // Reset transport memory from HMI10
      HMI10ResetSeq { ExternalAccessible := 'False'; ExternalVisible := 'False'; ExternalWritable := 'False'} : Bool;   // Reset sequence from HMI10
      HMI10CycleFinished { ExternalAccessible := 'False'; ExternalVisible := 'False'; ExternalWritable := 'False'} : Bool;   // Cycle Finished from HMI10
      HMI10AlarmResetAck { ExternalAccessible := 'False'; ExternalVisible := 'False'; ExternalWritable := 'False'} : Bool;   // Alarm Reset acknowledge from HMI10
      HMIGlobalAutoSel { ExternalAccessible := 'False'; ExternalVisible := 'False'; ExternalWritable := 'False'} : Bool;   // Auto selected on HMIxx
      HMIGlobalManualSel { ExternalAccessible := 'False'; ExternalVisible := 'False'; ExternalWritable := 'False'} : Bool;   // Manual selected on HMIxx
      HMIHomeRunRedo { ExternalAccessible := 'False'; ExternalVisible := 'False'; ExternalWritable := 'False'} : Bool;   // Redo after homerun from HMI
      HMIHomeRunWorkDone { ExternalAccessible := 'False'; ExternalVisible := 'False'; ExternalWritable := 'False'} : Bool;   // WorkDone after homerun from HMI
      LockManualTimeout { ExternalAccessible := 'False'; ExternalVisible := 'False'; ExternalWritable := 'False'} : Bool;   // Lock manual button timeout
      AllHmiAutoSel { ExternalAccessible := 'False'; ExternalVisible := 'False'; ExternalWritable := 'False'} : Bool;   // All Hmi Auto selected
      AlarmResetPBSel { ExternalAccessible := 'False'; ExternalVisible := 'False'; ExternalWritable := 'False'} : Bool;   // Alarm reset is activated
      AlarmResetPBSelReset { ExternalAccessible := 'False'; ExternalVisible := 'False'; ExternalWritable := 'False'} : Bool;   // Reset AlarmResetPBSel after predefined time
      AlarmResetPBSelResetPE { ExternalAccessible := 'False'; ExternalVisible := 'False'; ExternalWritable := 'False'} : Bool;   // Positive edge of AlarmResetPbSelReset
      StartPBSel { ExternalAccessible := 'False'; ExternalVisible := 'False'; ExternalWritable := 'False'} : Bool;   // Summary of the Start push buttons
      AutoSel { ExternalAccessible := 'False'; ExternalVisible := 'False'; ExternalWritable := 'False'} : Bool;   // Auto selected
      HMIStartPE { ExternalAccessible := 'False'; ExternalVisible := 'False'; ExternalWritable := 'False'} : Bool;   // Positive edge on start button from HMI
      HMIResetTMPE { ExternalAccessible := 'False'; ExternalVisible := 'False'; ExternalWritable := 'False'} : Bool;   // Positive edge on ResetTM button from HMI
      HMIResetSeqPE { ExternalAccessible := 'False'; ExternalVisible := 'False'; ExternalWritable := 'False'} : Bool;   // Positive edge on ResetSeq button from HMI
      HMIAlarmResetAckPE { ExternalAccessible := 'False'; ExternalVisible := 'False'; ExternalWritable := 'False'} : Bool;   // Positive edge on AlarmResetAck button from HMI
      HMILockManualPE { ExternalAccessible := 'False'; ExternalVisible := 'False'; ExternalWritable := 'False'} : Bool;   // Positive edge on LockManual button from HMI
      PBSetSel { ExternalAccessible := 'False'; ExternalVisible := 'False'; ExternalWritable := 'False'} : Bool;   // Set selected
      PBResetSel { ExternalAccessible := 'False'; ExternalVisible := 'False'; ExternalWritable := 'False'} : Bool;   // Reset selected
      CheckHMIActive { ExternalAccessible := 'False'; ExternalVisible := 'False'; ExternalWritable := 'False'} : Bool;   // Check Active HMI
      ActiveHMI { ExternalAccessible := 'False'; ExternalVisible := 'False'; ExternalWritable := 'False'} : Int;   // Help memory for Active HMI
      LockManualSec { ExternalAccessible := 'False'; ExternalVisible := 'False'; ExternalWritable := 'False'} : DInt;   // Lock manual on for xxx milliesec
      LockManualMillieSec { ExternalAccessible := 'False'; ExternalVisible := 'False'; ExternalWritable := 'False'} : DInt;   // Converted value
      TimerLockManValue { ExternalAccessible := 'False'; ExternalVisible := 'False'; ExternalWritable := 'False'} : DInt;   // Timer value
   END_VAR
   VAR
      TimerLockMan { ExternalAccessible := 'False'; ExternalVisible := 'False'; ExternalWritable := 'False'; S7_SetPoint := 'True'} : "LTimer";   // Timer on Lock manual
      TimerAlarmResetPB { ExternalAccessible := 'False'; ExternalVisible := 'False'; ExternalWritable := 'False'; S7_SetPoint := 'True'} : "LTimer";   // Timer on alarm reset
   END_VAR
   VAR DB_SPECIFIC
      CheckActiveHMI { ExternalAccessible := 'False'; ExternalVisible := 'False'; ExternalWritable := 'False'; S7_SetPoint := 'True'} : TP_TIME;   // Timer
      CheckActiveHMI_1 { ExternalAccessible := 'False'; ExternalVisible := 'False'; ExternalWritable := 'False'; S7_SetPoint := 'True'} : TP_TIME;   // Timer
      CheckActiveHMI_2 { ExternalAccessible := 'False'; ExternalVisible := 'False'; ExternalWritable := 'False'; S7_SetPoint := 'True'} : TON_TIME;   // Timer
      CheckActiveHMI_3 { ExternalAccessible := 'False'; ExternalVisible := 'False'; ExternalWritable := 'False'; S7_SetPoint := 'True'} : TON_TIME;   // Timer
      Edge { ExternalAccessible := 'False'; ExternalVisible := 'False'; ExternalWritable := 'False'; S7_SetPoint := 'True'} : Array[1..30] of Bool;
   END_VAR
   VAR_TEMP
      PHMI1AutoSel : Bool;   // Pulse Auto selected HMI1
      PHMI2AutoSel : Bool;   // Pulse Auto selected HMI2
      PHMI3AutoSel : Bool;   // Pulse Auto selected HMI3
      PHMI4AutoSel : Bool;   // Pulse Auto selected HMI4
      PHMI5AutoSel : Bool;   // Pulse Auto selected HMI5
      PHMI6AutoSel : Bool;   // Pulse Auto selected HMI6
      PHMI7AutoSel : Bool;   // Pulse Auto selected HMI7
      PHMI8AutoSel : Bool;   // Pulse Auto selected HMI8
      PHMI9AutoSel : Bool;   // Pulse Auto selected HMI9
      PHMI10AutoSel : Bool;   // Pulse Auto selected HMI10
      LockManualTime : Int;   // Lock manual time
      LockManualTimeInt : Int;   // Lock manual time
      LockManualTimeDInt : DInt;   // Lock manual time
   END_VAR
   VAR_TEMP   // added for the SCL form of the ladder/FBD networks
      _w1 : Bool;
      _w2 : Bool;
      _w3 : Bool;
      _w4 : Bool;
      _w5 : Bool;
      _w6 : Bool;
      _w7 : Bool;
      _w8 : Bool;
      _w9 : Bool;
      _w10 : Bool;
   END_VAR
BEGIN

REGION Network 1: ---------------------------------------------------------- Human Machine Interface 1 ----------------------------------------------------------
END_REGION

REGION Network 2: **** 1 - Inputs **** HMI-1 : Extract the modeselection from HMI
   // Extract the modeselection from HMI 1
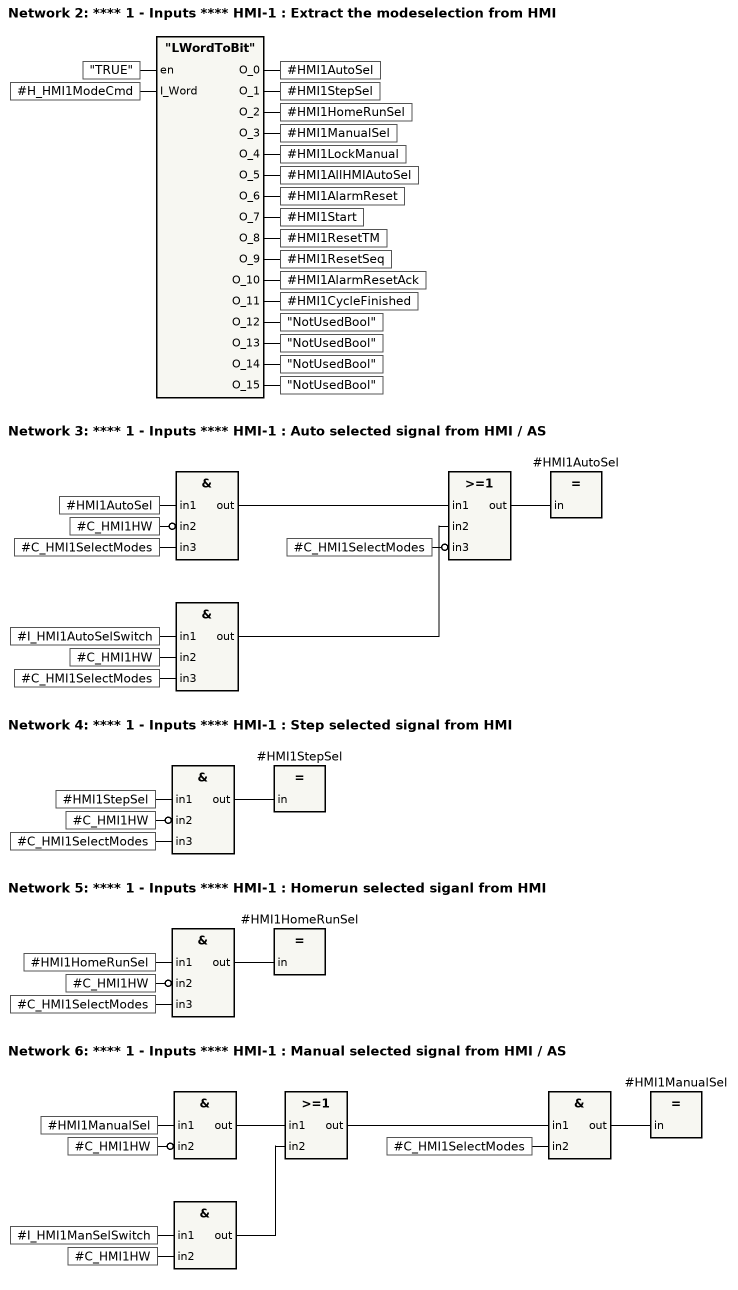
   IF "TRUE" THEN
       "LWordToBit"(I_Word := #H_HMI1ModeCmd,
                    O_0 => #HMI1AutoSel,
                    O_1 => #HMI1StepSel,
                    O_2 => #HMI1HomeRunSel,
                    O_3 => #HMI1ManualSel,
                    O_4 => #HMI1LockManual,
                    O_5 => #HMI1AllHMIAutoSel,
                    O_6 => #HMI1AlarmReset,
                    O_7 => #HMI1Start,
                    O_8 => #HMI1ResetTM,
                    O_9 => #HMI1ResetSeq,
                    O_10 => #HMI1AlarmResetAck,
                    O_11 => #HMI1CycleFinished,
                    O_12 => "NotUsedBool",
                    O_13 => "NotUsedBool",
                    O_14 => "NotUsedBool",
                    O_15 => "NotUsedBool");
   END_IF;
END_REGION

REGION Network 3: **** 1 - Inputs **** HMI-1 : Auto selected signal from HMI / AS
   #HMI1AutoSel := (#HMI1AutoSel AND NOT #C_HMI1HW AND #C_HMI1SelectModes) OR (#I_HMI1AutoSelSwitch AND #C_HMI1HW AND #C_HMI1SelectModes) OR NOT #C_HMI1SelectModes;
END_REGION

REGION Network 4: **** 1 - Inputs **** HMI-1 : Step selected signal from HMI
   #HMI1StepSel := #HMI1StepSel AND NOT #C_HMI1HW AND #C_HMI1SelectModes;
END_REGION

REGION Network 5: **** 1 - Inputs **** HMI-1 : Homerun selected siganl from HMI
   #HMI1HomeRunSel := #HMI1HomeRunSel AND NOT #C_HMI1HW AND #C_HMI1SelectModes;
END_REGION

REGION Network 6: **** 1 - Inputs **** HMI-1 : Manual selected signal from HMI / AS
   #HMI1ManualSel := ((#HMI1ManualSel AND NOT #C_HMI1HW) OR (#I_HMI1ManSelSwitch AND #C_HMI1HW)) AND #C_HMI1SelectModes;
END_REGION

REGION Network 7: ---------------------------------------------------------- Human Machine Interface 2 ----------------------------------------------------------
END_REGION

REGION Network 8: **** 1 - Inputs **** HMI-2 : Extract the modeselection from HMI
   // Extract the modeselection from HMI 2
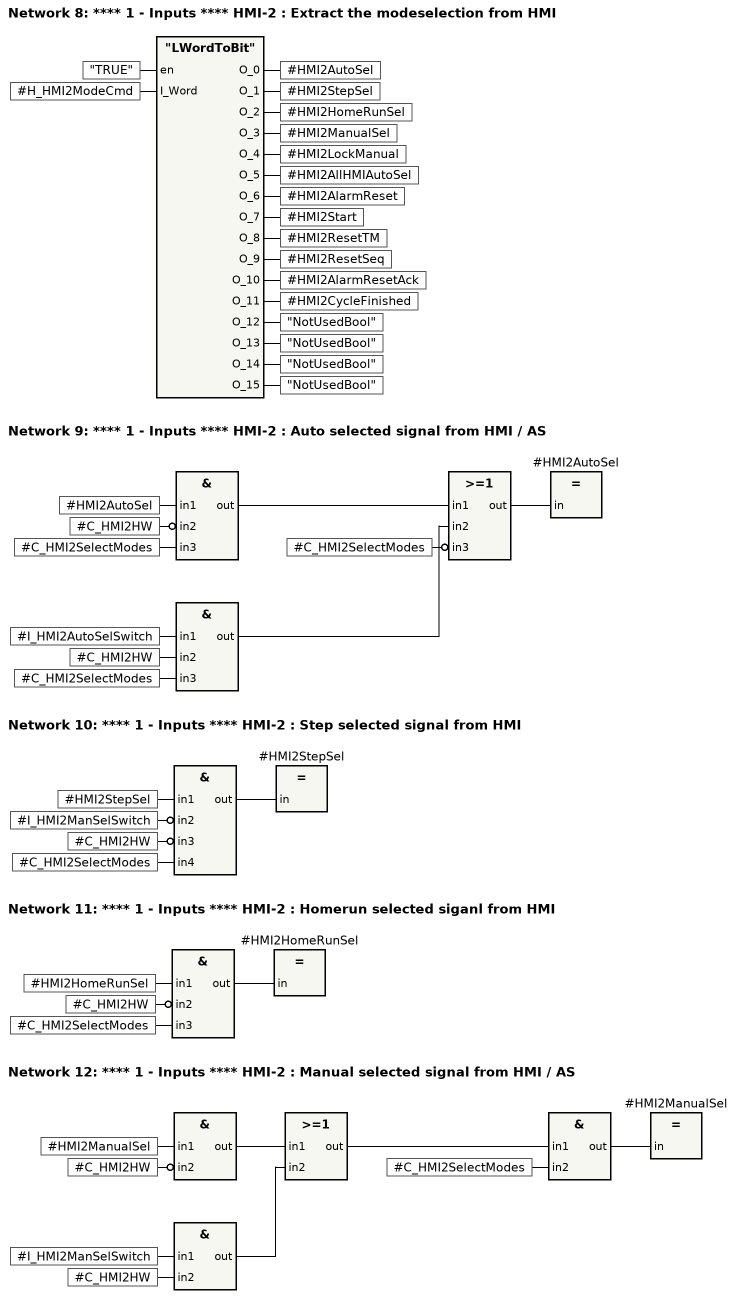
   IF "TRUE" THEN
       "LWordToBit"(I_Word := #H_HMI2ModeCmd,
                    O_0 => #HMI2AutoSel,
                    O_1 => #HMI2StepSel,
                    O_2 => #HMI2HomeRunSel,
                    O_3 => #HMI2ManualSel,
                    O_4 => #HMI2LockManual,
                    O_5 => #HMI2AllHMIAutoSel,
                    O_6 => #HMI2AlarmReset,
                    O_7 => #HMI2Start,
                    O_8 => #HMI2ResetTM,
                    O_9 => #HMI2ResetSeq,
                    O_10 => #HMI2AlarmResetAck,
                    O_11 => #HMI2CycleFinished,
                    O_12 => "NotUsedBool",
                    O_13 => "NotUsedBool",
                    O_14 => "NotUsedBool",
                    O_15 => "NotUsedBool");
   END_IF;
END_REGION

REGION Network 9: **** 1 - Inputs **** HMI-2 : Auto selected signal from HMI / AS
   #HMI2AutoSel := (#HMI2AutoSel AND NOT #C_HMI2HW AND #C_HMI2SelectModes) OR (#I_HMI2AutoSelSwitch AND #C_HMI2HW AND #C_HMI2SelectModes) OR NOT #C_HMI2SelectModes;
END_REGION

REGION Network 10: **** 1 - Inputs **** HMI-2 : Step selected signal from HMI
   #HMI2StepSel := #HMI2StepSel AND NOT #I_HMI2ManSelSwitch AND NOT #C_HMI2HW AND #C_HMI2SelectModes;
END_REGION

REGION Network 11: **** 1 - Inputs **** HMI-2 : Homerun selected siganl from HMI
   #HMI2HomeRunSel := #HMI2HomeRunSel AND NOT #C_HMI2HW AND #C_HMI2SelectModes;
END_REGION

REGION Network 12: **** 1 - Inputs **** HMI-2 : Manual selected signal from HMI / AS
   #HMI2ManualSel := ((#HMI2ManualSel AND NOT #C_HMI2HW) OR (#I_HMI2ManSelSwitch AND #C_HMI2HW)) AND #C_HMI2SelectModes;
END_REGION

REGION Network 13: ---------------------------------------------------------- Human Machine Interface 3 ----------------------------------------------------------
END_REGION

REGION Network 14: **** 1 - Inputs **** HMI-3 : Extract the modeselection from HMI
   // Extract the modeselection from HMI 3
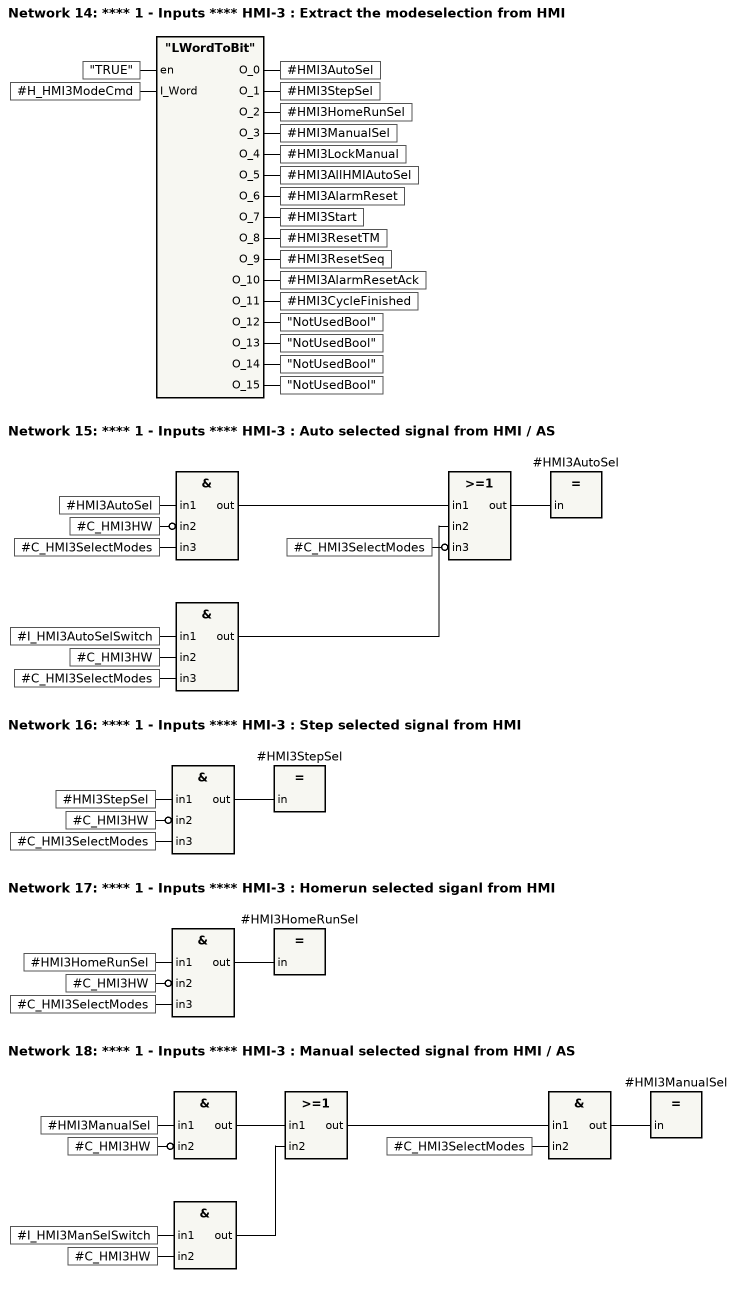
   IF "TRUE" THEN
       "LWordToBit"(I_Word := #H_HMI3ModeCmd,
                    O_0 => #HMI3AutoSel,
                    O_1 => #HMI3StepSel,
                    O_2 => #HMI3HomeRunSel,
                    O_3 => #HMI3ManualSel,
                    O_4 => #HMI3LockManual,
                    O_5 => #HMI3AllHMIAutoSel,
                    O_6 => #HMI3AlarmReset,
                    O_7 => #HMI3Start,
                    O_8 => #HMI3ResetTM,
                    O_9 => #HMI3ResetSeq,
                    O_10 => #HMI3AlarmResetAck,
                    O_11 => #HMI3CycleFinished,
                    O_12 => "NotUsedBool",
                    O_13 => "NotUsedBool",
                    O_14 => "NotUsedBool",
                    O_15 => "NotUsedBool");
   END_IF;
END_REGION

REGION Network 15: **** 1 - Inputs **** HMI-3 : Auto selected signal from HMI / AS
   #HMI3AutoSel := (#HMI3AutoSel AND NOT #C_HMI3HW AND #C_HMI3SelectModes) OR (#I_HMI3AutoSelSwitch AND #C_HMI3HW AND #C_HMI3SelectModes) OR NOT #C_HMI3SelectModes;
END_REGION

REGION Network 16: **** 1 - Inputs **** HMI-3 : Step selected signal from HMI
   #HMI3StepSel := #HMI3StepSel AND NOT #C_HMI3HW AND #C_HMI3SelectModes;
END_REGION

REGION Network 17: **** 1 - Inputs **** HMI-3 : Homerun selected siganl from HMI
   #HMI3HomeRunSel := #HMI3HomeRunSel AND NOT #C_HMI3HW AND #C_HMI3SelectModes;
END_REGION

REGION Network 18: **** 1 - Inputs **** HMI-3 : Manual selected signal from HMI / AS
   #HMI3ManualSel := ((#HMI3ManualSel AND NOT #C_HMI3HW) OR (#I_HMI3ManSelSwitch AND #C_HMI3HW)) AND #C_HMI3SelectModes;
END_REGION

REGION Network 19: ---------------------------------------------------------- Human Machine Interface 4 ----------------------------------------------------------
END_REGION

REGION Network 20: **** 1 - Inputs **** HMI-4 : Extract the modeselection from HMI
   // Extract the modeselection from HMI 4
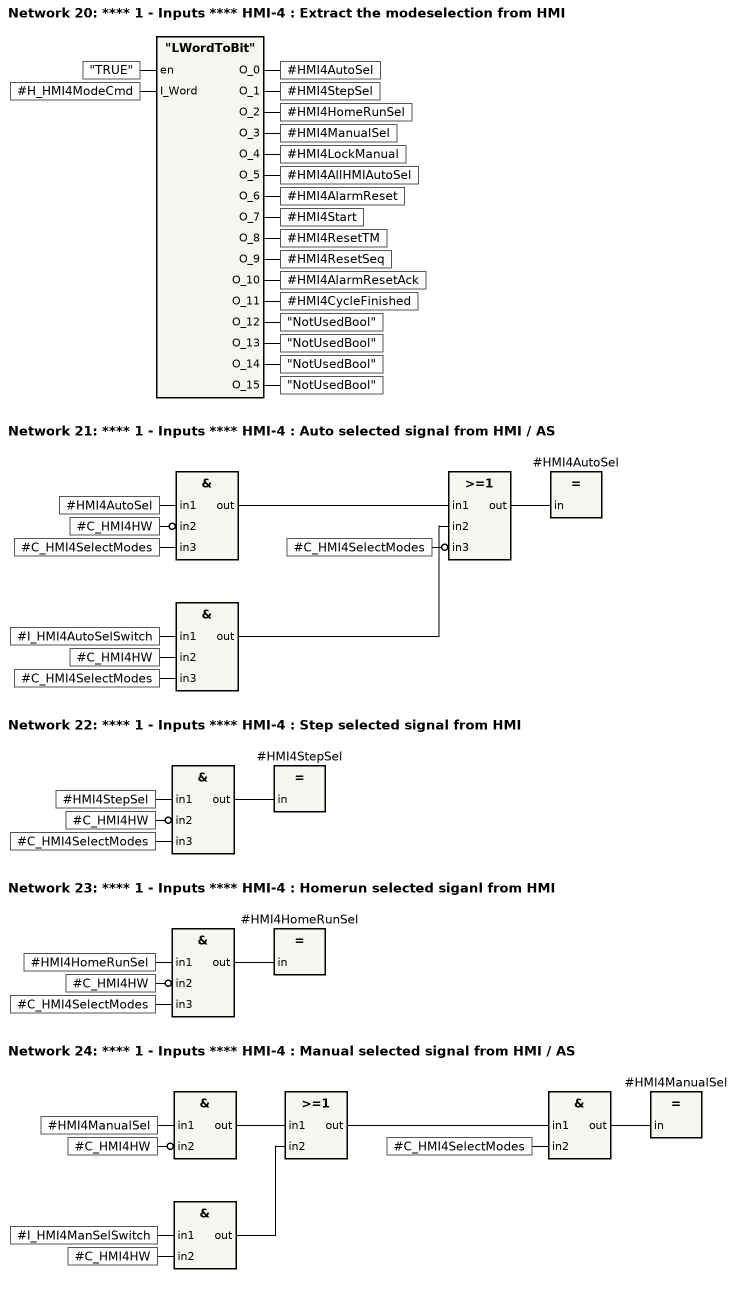
   IF "TRUE" THEN
       "LWordToBit"(I_Word := #H_HMI4ModeCmd,
                    O_0 => #HMI4AutoSel,
                    O_1 => #HMI4StepSel,
                    O_2 => #HMI4HomeRunSel,
                    O_3 => #HMI4ManualSel,
                    O_4 => #HMI4LockManual,
                    O_5 => #HMI4AllHMIAutoSel,
                    O_6 => #HMI4AlarmReset,
                    O_7 => #HMI4Start,
                    O_8 => #HMI4ResetTM,
                    O_9 => #HMI4ResetSeq,
                    O_10 => #HMI4AlarmResetAck,
                    O_11 => #HMI4CycleFinished,
                    O_12 => "NotUsedBool",
                    O_13 => "NotUsedBool",
                    O_14 => "NotUsedBool",
                    O_15 => "NotUsedBool");
   END_IF;
END_REGION

REGION Network 21: **** 1 - Inputs **** HMI-4 : Auto selected signal from HMI / AS
   #HMI4AutoSel := (#HMI4AutoSel AND NOT #C_HMI4HW AND #C_HMI4SelectModes) OR (#I_HMI4AutoSelSwitch AND #C_HMI4HW AND #C_HMI4SelectModes) OR NOT #C_HMI4SelectModes;
END_REGION

REGION Network 22: **** 1 - Inputs **** HMI-4 : Step selected signal from HMI
   #HMI4StepSel := #HMI4StepSel AND NOT #C_HMI4HW AND #C_HMI4SelectModes;
END_REGION

REGION Network 23: **** 1 - Inputs **** HMI-4 : Homerun selected siganl from HMI
   #HMI4HomeRunSel := #HMI4HomeRunSel AND NOT #C_HMI4HW AND #C_HMI4SelectModes;
END_REGION

REGION Network 24: **** 1 - Inputs **** HMI-4 : Manual selected signal from HMI / AS
   #HMI4ManualSel := ((#HMI4ManualSel AND NOT #C_HMI4HW) OR (#I_HMI4ManSelSwitch AND #C_HMI4HW)) AND #C_HMI4SelectModes;
END_REGION

REGION Network 25: ---------------------------------------------------------- Human Machine Interface 5 ----------------------------------------------------------
END_REGION

REGION Network 26: **** 1 - Inputs **** HMI-5 : Extract the modeselection from HMI
   // Extract the modeselection from HMI 5
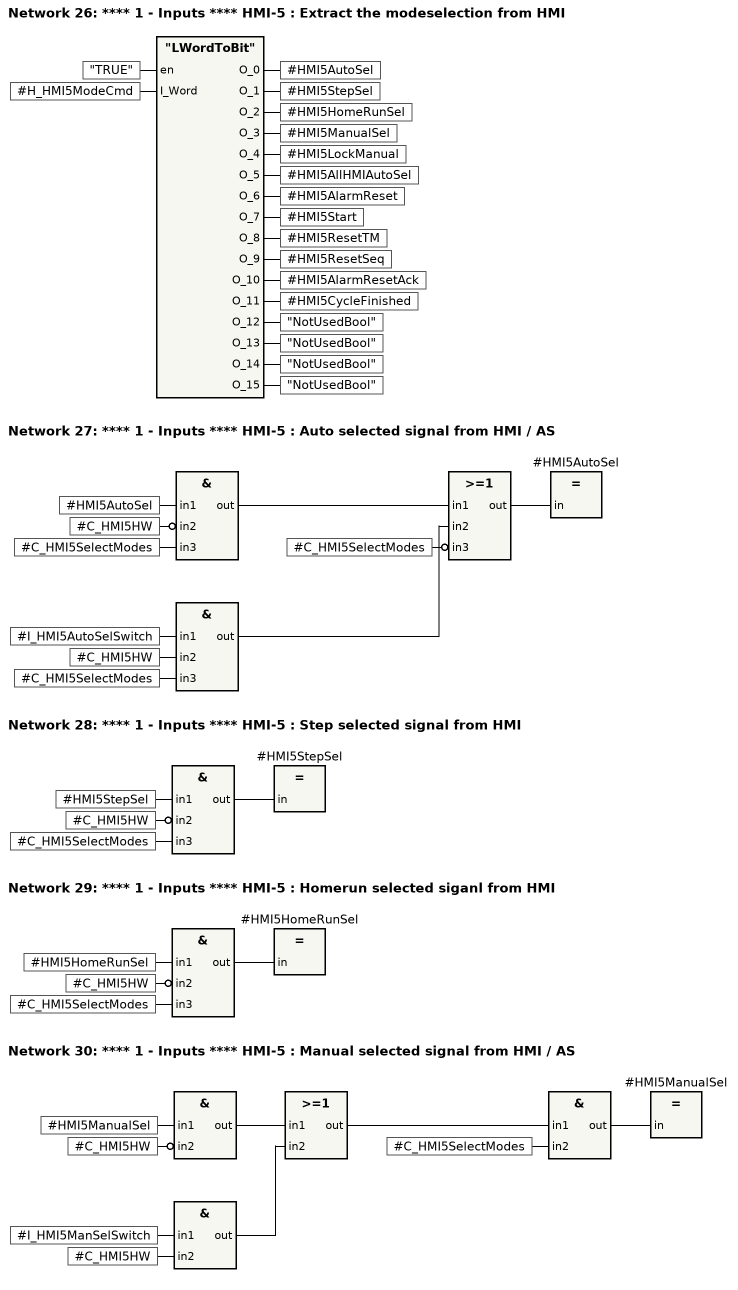
   IF "TRUE" THEN
       "LWordToBit"(I_Word := #H_HMI5ModeCmd,
                    O_0 => #HMI5AutoSel,
                    O_1 => #HMI5StepSel,
                    O_2 => #HMI5HomeRunSel,
                    O_3 => #HMI5ManualSel,
                    O_4 => #HMI5LockManual,
                    O_5 => #HMI5AllHMIAutoSel,
                    O_6 => #HMI5AlarmReset,
                    O_7 => #HMI5Start,
                    O_8 => #HMI5ResetTM,
                    O_9 => #HMI5ResetSeq,
                    O_10 => #HMI5AlarmResetAck,
                    O_11 => #HMI5CycleFinished,
                    O_12 => "NotUsedBool",
                    O_13 => "NotUsedBool",
                    O_14 => "NotUsedBool",
                    O_15 => "NotUsedBool");
   END_IF;
END_REGION

REGION Network 27: **** 1 - Inputs **** HMI-5 : Auto selected signal from HMI / AS
   #HMI5AutoSel := (#HMI5AutoSel AND NOT #C_HMI5HW AND #C_HMI5SelectModes) OR (#I_HMI5AutoSelSwitch AND #C_HMI5HW AND #C_HMI5SelectModes) OR NOT #C_HMI5SelectModes;
END_REGION

REGION Network 28: **** 1 - Inputs **** HMI-5 : Step selected signal from HMI
   #HMI5StepSel := #HMI5StepSel AND NOT #C_HMI5HW AND #C_HMI5SelectModes;
END_REGION

REGION Network 29: **** 1 - Inputs **** HMI-5 : Homerun selected siganl from HMI
   #HMI5HomeRunSel := #HMI5HomeRunSel AND NOT #C_HMI5HW AND #C_HMI5SelectModes;
END_REGION

REGION Network 30: **** 1 - Inputs **** HMI-5 : Manual selected signal from HMI / AS
   #HMI5ManualSel := ((#HMI5ManualSel AND NOT #C_HMI5HW) OR (#I_HMI5ManSelSwitch AND #C_HMI5HW)) AND #C_HMI5SelectModes;
END_REGION

REGION Network 31: ---------------------------------------------------------- Human Machine Interface 6 ----------------------------------------------------------
END_REGION

REGION Network 32: **** 1 - Inputs **** HMI-6 : Extract the modeselection from HMI
   // Extract the modeselection from HMI 6
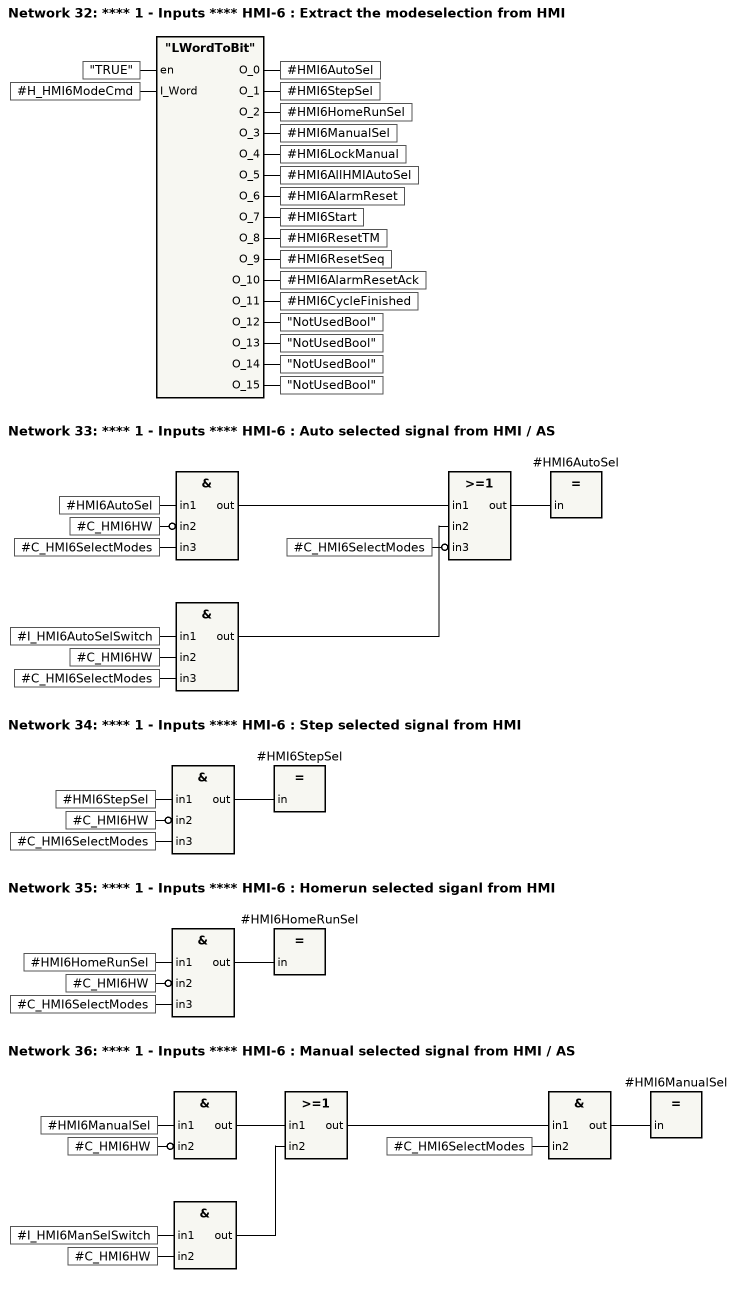
   IF "TRUE" THEN
       "LWordToBit"(I_Word := #H_HMI6ModeCmd,
                    O_0 => #HMI6AutoSel,
                    O_1 => #HMI6StepSel,
                    O_2 => #HMI6HomeRunSel,
                    O_3 => #HMI6ManualSel,
                    O_4 => #HMI6LockManual,
                    O_5 => #HMI6AllHMIAutoSel,
                    O_6 => #HMI6AlarmReset,
                    O_7 => #HMI6Start,
                    O_8 => #HMI6ResetTM,
                    O_9 => #HMI6ResetSeq,
                    O_10 => #HMI6AlarmResetAck,
                    O_11 => #HMI6CycleFinished,
                    O_12 => "NotUsedBool",
                    O_13 => "NotUsedBool",
                    O_14 => "NotUsedBool",
                    O_15 => "NotUsedBool");
   END_IF;
END_REGION

REGION Network 33: **** 1 - Inputs **** HMI-6 : Auto selected signal from HMI / AS
   #HMI6AutoSel := (#HMI6AutoSel AND NOT #C_HMI6HW AND #C_HMI6SelectModes) OR (#I_HMI6AutoSelSwitch AND #C_HMI6HW AND #C_HMI6SelectModes) OR NOT #C_HMI6SelectModes;
END_REGION

REGION Network 34: **** 1 - Inputs **** HMI-6 : Step selected signal from HMI
   #HMI6StepSel := #HMI6StepSel AND NOT #C_HMI6HW AND #C_HMI6SelectModes;
END_REGION

REGION Network 35: **** 1 - Inputs **** HMI-6 : Homerun selected siganl from HMI
   #HMI6HomeRunSel := #HMI6HomeRunSel AND NOT #C_HMI6HW AND #C_HMI6SelectModes;
END_REGION

REGION Network 36: **** 1 - Inputs **** HMI-6 : Manual selected signal from HMI / AS
   #HMI6ManualSel := ((#HMI6ManualSel AND NOT #C_HMI6HW) OR (#I_HMI6ManSelSwitch AND #C_HMI6HW)) AND #C_HMI6SelectModes;
END_REGION

REGION Network 37: ---------------------------------------------------------- Human Machine Interface 7 ----------------------------------------------------------
END_REGION

REGION Network 38: **** 1 - Inputs **** HMI-7 : Extract the modeselection from HMI
   // Extract the modeselection from HMI 7
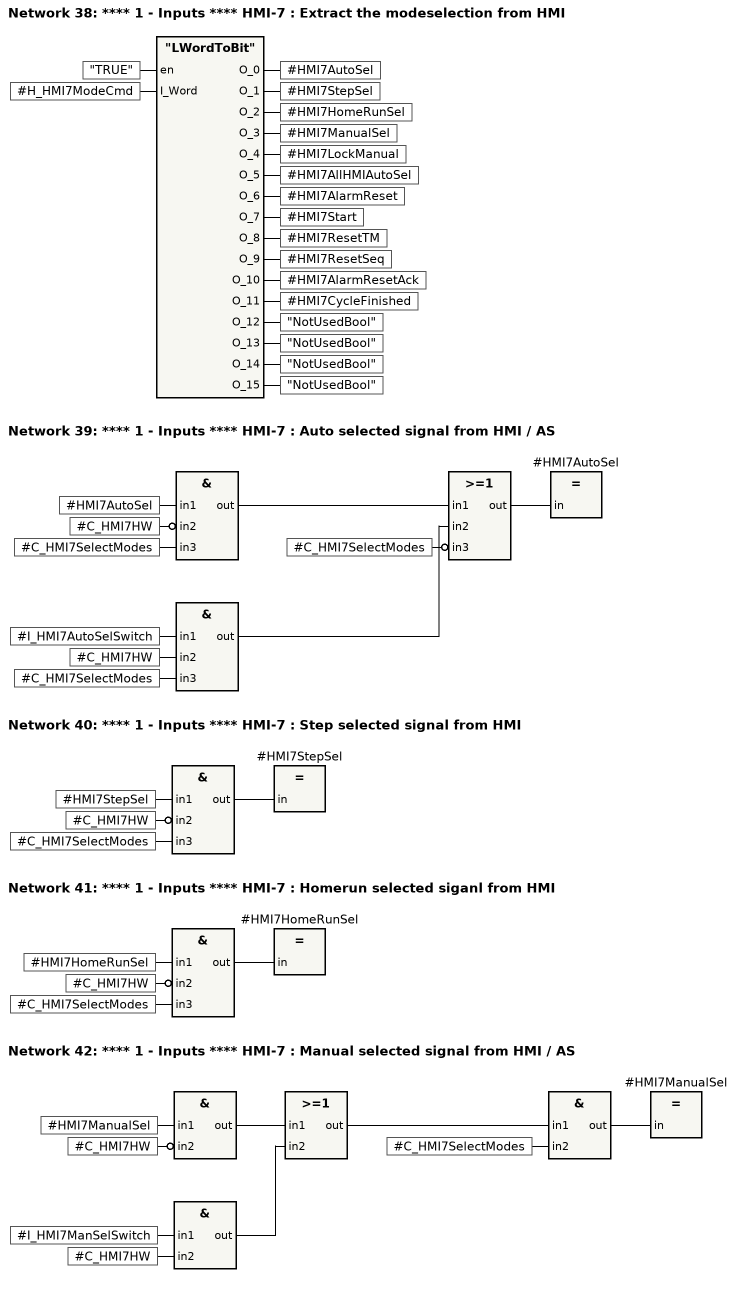
   IF "TRUE" THEN
       "LWordToBit"(I_Word := #H_HMI7ModeCmd,
                    O_0 => #HMI7AutoSel,
                    O_1 => #HMI7StepSel,
                    O_2 => #HMI7HomeRunSel,
                    O_3 => #HMI7ManualSel,
                    O_4 => #HMI7LockManual,
                    O_5 => #HMI7AllHMIAutoSel,
                    O_6 => #HMI7AlarmReset,
                    O_7 => #HMI7Start,
                    O_8 => #HMI7ResetTM,
                    O_9 => #HMI7ResetSeq,
                    O_10 => #HMI7AlarmResetAck,
                    O_11 => #HMI7CycleFinished,
                    O_12 => "NotUsedBool",
                    O_13 => "NotUsedBool",
                    O_14 => "NotUsedBool",
                    O_15 => "NotUsedBool");
   END_IF;
END_REGION

REGION Network 39: **** 1 - Inputs **** HMI-7 : Auto selected signal from HMI / AS
   #HMI7AutoSel := (#HMI7AutoSel AND NOT #C_HMI7HW AND #C_HMI7SelectModes) OR (#I_HMI7AutoSelSwitch AND #C_HMI7HW AND #C_HMI7SelectModes) OR NOT #C_HMI7SelectModes;
END_REGION

REGION Network 40: **** 1 - Inputs **** HMI-7 : Step selected signal from HMI
   #HMI7StepSel := #HMI7StepSel AND NOT #C_HMI7HW AND #C_HMI7SelectModes;
END_REGION

REGION Network 41: **** 1 - Inputs **** HMI-7 : Homerun selected siganl from HMI
   #HMI7HomeRunSel := #HMI7HomeRunSel AND NOT #C_HMI7HW AND #C_HMI7SelectModes;
END_REGION

REGION Network 42: **** 1 - Inputs **** HMI-7 : Manual selected signal from HMI / AS
   #HMI7ManualSel := ((#HMI7ManualSel AND NOT #C_HMI7HW) OR (#I_HMI7ManSelSwitch AND #C_HMI7HW)) AND #C_HMI7SelectModes;
END_REGION

REGION Network 43: ---------------------------------------------------------- Human Machine Interface 8 ----------------------------------------------------------
END_REGION

REGION Network 44: **** 1 - Inputs **** HMI-8 : Extract the modeselection from HMI
   // Extract the modeselection from HMI 8
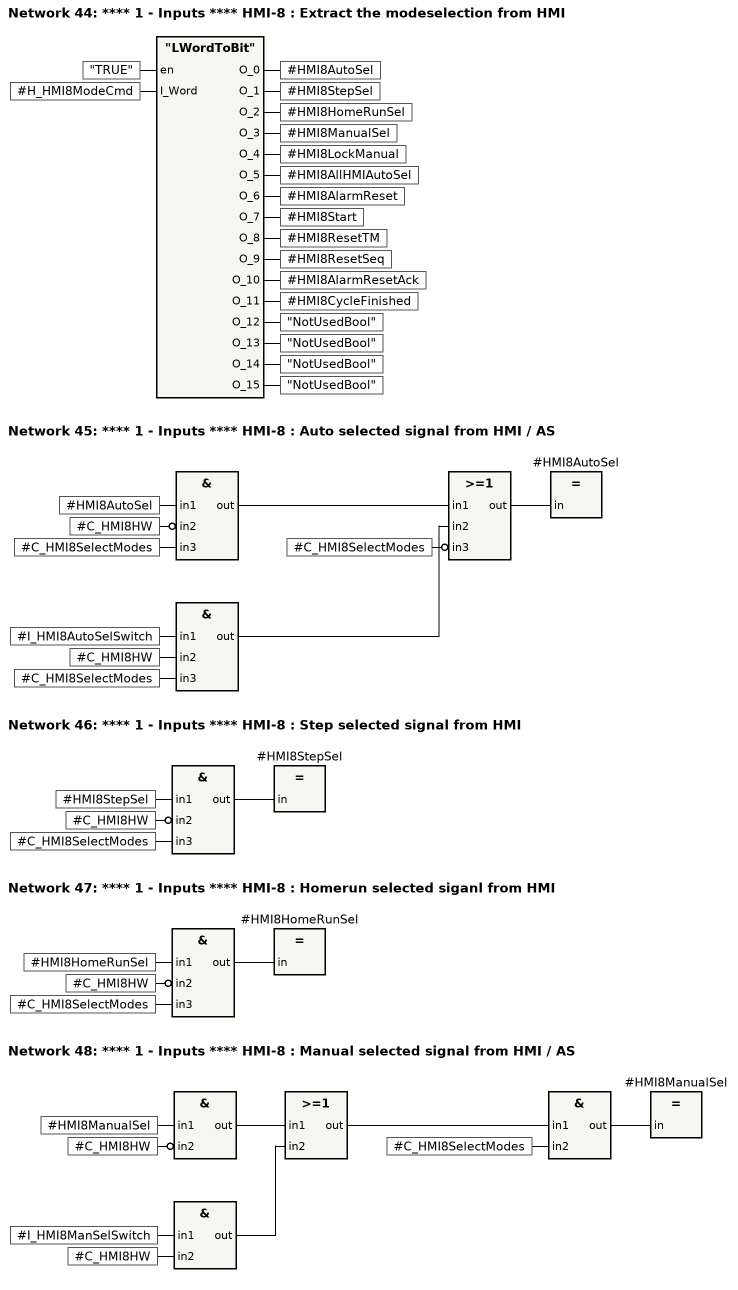
   IF "TRUE" THEN
       "LWordToBit"(I_Word := #H_HMI8ModeCmd,
                    O_0 => #HMI8AutoSel,
                    O_1 => #HMI8StepSel,
                    O_2 => #HMI8HomeRunSel,
                    O_3 => #HMI8ManualSel,
                    O_4 => #HMI8LockManual,
                    O_5 => #HMI8AllHMIAutoSel,
                    O_6 => #HMI8AlarmReset,
                    O_7 => #HMI8Start,
                    O_8 => #HMI8ResetTM,
                    O_9 => #HMI8ResetSeq,
                    O_10 => #HMI8AlarmResetAck,
                    O_11 => #HMI8CycleFinished,
                    O_12 => "NotUsedBool",
                    O_13 => "NotUsedBool",
                    O_14 => "NotUsedBool",
                    O_15 => "NotUsedBool");
   END_IF;
END_REGION

REGION Network 45: **** 1 - Inputs **** HMI-8 : Auto selected signal from HMI / AS
   #HMI8AutoSel := (#HMI8AutoSel AND NOT #C_HMI8HW AND #C_HMI8SelectModes) OR (#I_HMI8AutoSelSwitch AND #C_HMI8HW AND #C_HMI8SelectModes) OR NOT #C_HMI8SelectModes;
END_REGION

REGION Network 46: **** 1 - Inputs **** HMI-8 : Step selected signal from HMI
   #HMI8StepSel := #HMI8StepSel AND NOT #C_HMI8HW AND #C_HMI8SelectModes;
END_REGION

REGION Network 47: **** 1 - Inputs **** HMI-8 : Homerun selected siganl from HMI
   #HMI8HomeRunSel := #HMI8HomeRunSel AND NOT #C_HMI8HW AND #C_HMI8SelectModes;
END_REGION

REGION Network 48: **** 1 - Inputs **** HMI-8 : Manual selected signal from HMI / AS
   #HMI8ManualSel := ((#HMI8ManualSel AND NOT #C_HMI8HW) OR (#I_HMI8ManSelSwitch AND #C_HMI8HW)) AND #C_HMI8SelectModes;
END_REGION

REGION Network 49: ---------------------------------------------------------- Human Machine Interface 9 ----------------------------------------------------------
END_REGION

REGION Network 50: **** 1 - Inputs **** HMI-9 : Extract the modeselection from HMI
   // Extract the modeselection from HMI 9
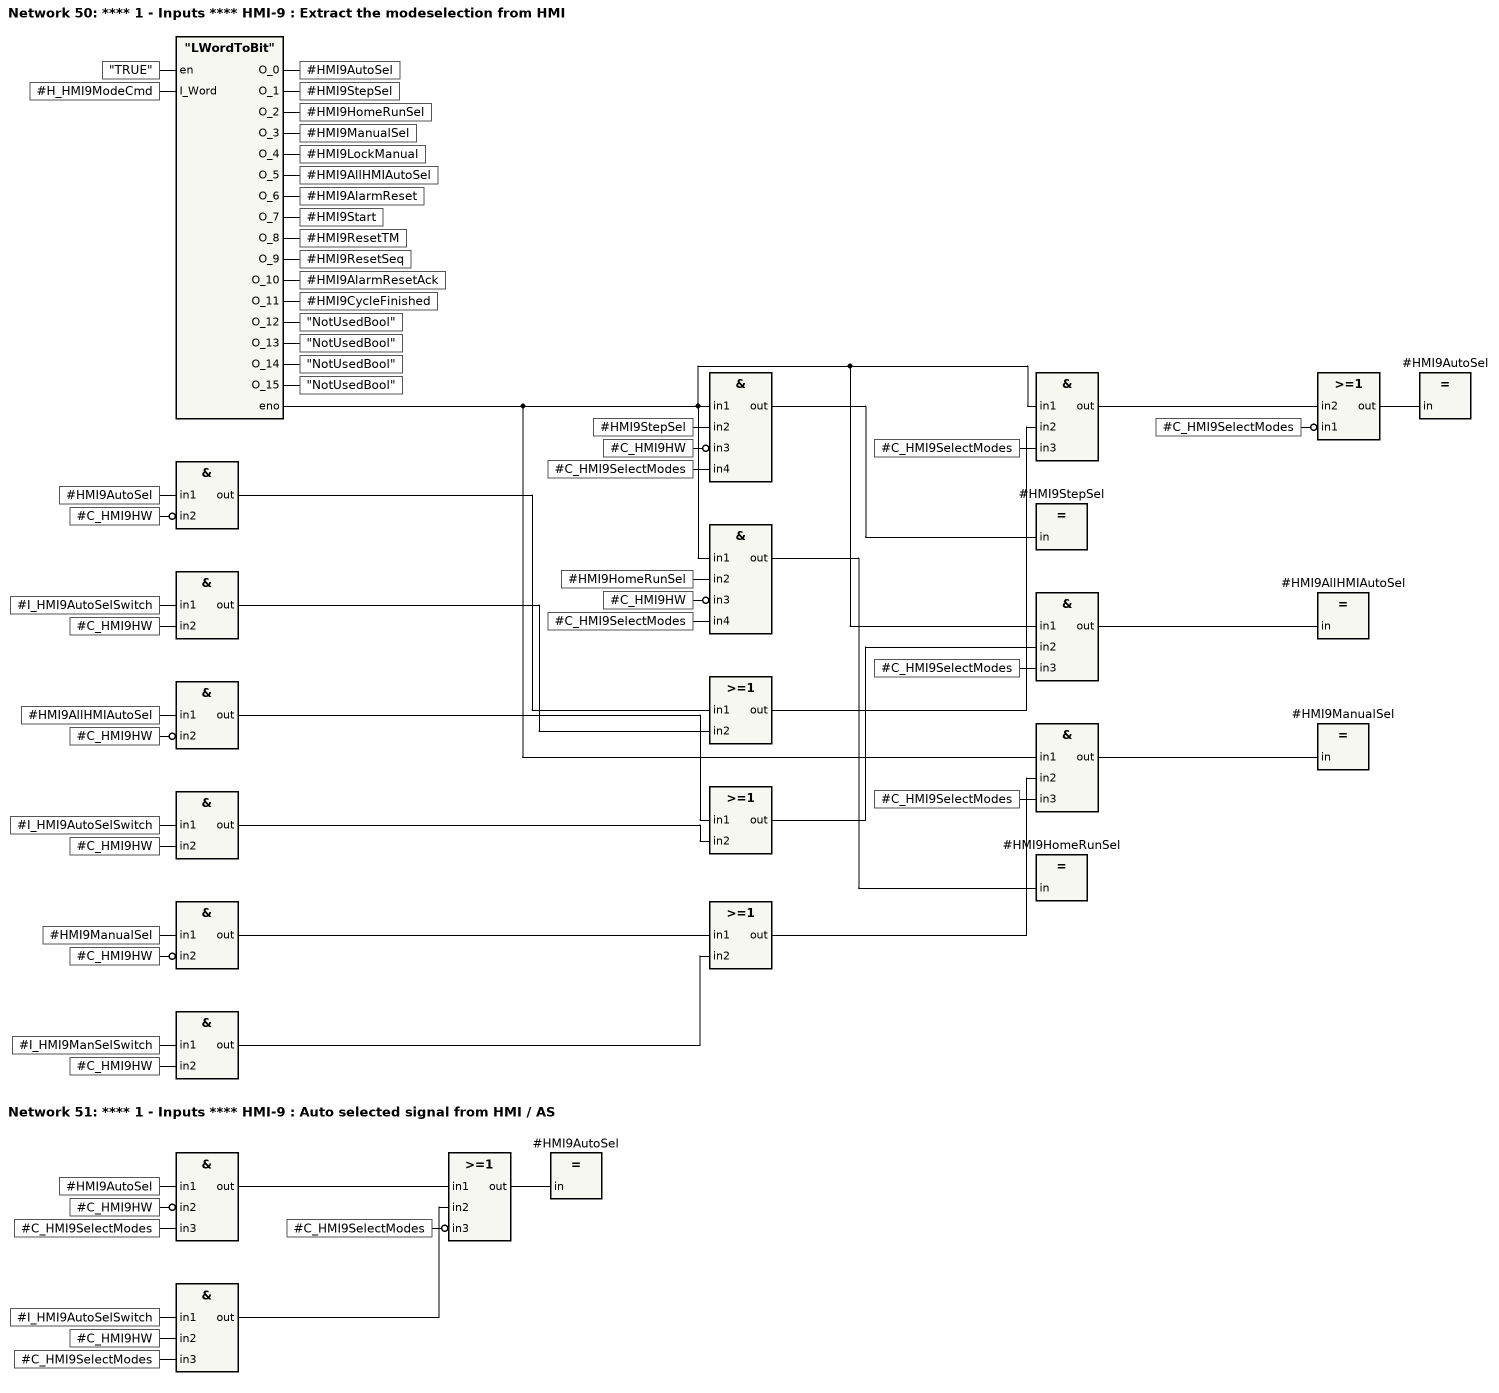
   "LWordToBit"(EN := "TRUE",
                I_Word := #H_HMI9ModeCmd,
                O_0 => #HMI9AutoSel,
                O_1 => #HMI9StepSel,
                O_2 => #HMI9HomeRunSel,
                O_3 => #HMI9ManualSel,
                O_4 => #HMI9LockManual,
                O_5 => #HMI9AllHMIAutoSel,
                O_6 => #HMI9AlarmReset,
                O_7 => #HMI9Start,
                O_8 => #HMI9ResetTM,
                O_9 => #HMI9ResetSeq,
                O_10 => #HMI9AlarmResetAck,
                O_11 => #HMI9CycleFinished,
                O_12 => "NotUsedBool",
                O_13 => "NotUsedBool",
                O_14 => "NotUsedBool",
                O_15 => "NotUsedBool",
                ENO => #_w1);
   #HMI9AutoSel := (#_w1 AND ((#HMI9AutoSel AND NOT #C_HMI9HW) OR (#I_HMI9AutoSelSwitch AND #C_HMI9HW)) AND #C_HMI9SelectModes) OR NOT #C_HMI9SelectModes;
   #HMI9StepSel := #_w1 AND #HMI9StepSel AND NOT #C_HMI9HW AND #C_HMI9SelectModes;
   #HMI9HomeRunSel := #_w1 AND #HMI9HomeRunSel AND NOT #C_HMI9HW AND #C_HMI9SelectModes;
   #HMI9AllHMIAutoSel := #_w1 AND ((#HMI9AllHMIAutoSel AND NOT #C_HMI9HW) OR (#I_HMI9AutoSelSwitch AND #C_HMI9HW)) AND #C_HMI9SelectModes;
   #HMI9ManualSel := #_w1 AND ((#HMI9ManualSel AND NOT #C_HMI9HW) OR (#I_HMI9ManSelSwitch AND #C_HMI9HW)) AND #C_HMI9SelectModes;
END_REGION

REGION Network 51: **** 1 - Inputs **** HMI-9 : Auto selected signal from HMI / AS
   #HMI9AutoSel := (#HMI9AutoSel AND NOT #C_HMI9HW AND #C_HMI9SelectModes) OR (#I_HMI9AutoSelSwitch AND #C_HMI9HW AND #C_HMI9SelectModes) OR NOT #C_HMI9SelectModes;
END_REGION

REGION Network 52: **** 1 - Inputs **** HMI-9 : Step selected signal from HMI
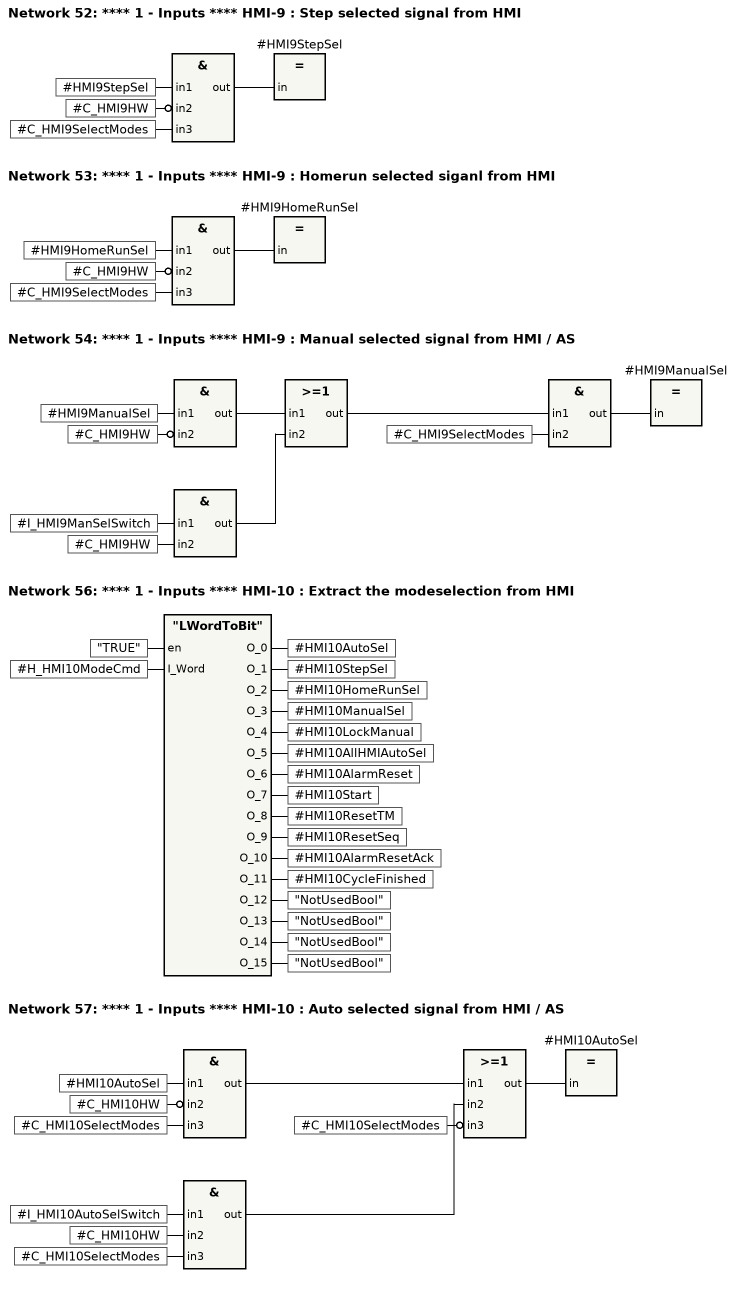
   #HMI9StepSel := #HMI9StepSel AND NOT #C_HMI9HW AND #C_HMI9SelectModes;
END_REGION

REGION Network 53: **** 1 - Inputs **** HMI-9 : Homerun selected siganl from HMI
   #HMI9HomeRunSel := #HMI9HomeRunSel AND NOT #C_HMI9HW AND #C_HMI9SelectModes;
END_REGION

REGION Network 54: **** 1 - Inputs **** HMI-9 : Manual selected signal from HMI / AS
   #HMI9ManualSel := ((#HMI9ManualSel AND NOT #C_HMI9HW) OR (#I_HMI9ManSelSwitch AND #C_HMI9HW)) AND #C_HMI9SelectModes;
END_REGION

REGION Network 55: ---------------------------------------------------------- Human Machine Interface 10 ----------------------------------------------------------
END_REGION

REGION Network 56: **** 1 - Inputs **** HMI-10 : Extract the modeselection from HMI
   // Extract the modeselection from HMI 10
   IF "TRUE" THEN
       "LWordToBit"(I_Word := #H_HMI10ModeCmd,
                    O_0 => #HMI10AutoSel,
                    O_1 => #HMI10StepSel,
                    O_2 => #HMI10HomeRunSel,
                    O_3 => #HMI10ManualSel,
                    O_4 => #HMI10LockManual,
                    O_5 => #HMI10AllHMIAutoSel,
                    O_6 => #HMI10AlarmReset,
                    O_7 => #HMI10Start,
                    O_8 => #HMI10ResetTM,
                    O_9 => #HMI10ResetSeq,
                    O_10 => #HMI10AlarmResetAck,
                    O_11 => #HMI10CycleFinished,
                    O_12 => "NotUsedBool",
                    O_13 => "NotUsedBool",
                    O_14 => "NotUsedBool",
                    O_15 => "NotUsedBool");
   END_IF;
END_REGION

REGION Network 57: **** 1 - Inputs **** HMI-10 : Auto selected signal from HMI / AS
   #HMI10AutoSel := (#HMI10AutoSel AND NOT #C_HMI10HW AND #C_HMI10SelectModes) OR (#I_HMI10AutoSelSwitch AND #C_HMI10HW AND #C_HMI10SelectModes) OR NOT #C_HMI10SelectModes;
END_REGION

REGION Network 58: **** 1 - Inputs **** HMI-10 : Step selected signal from HMI
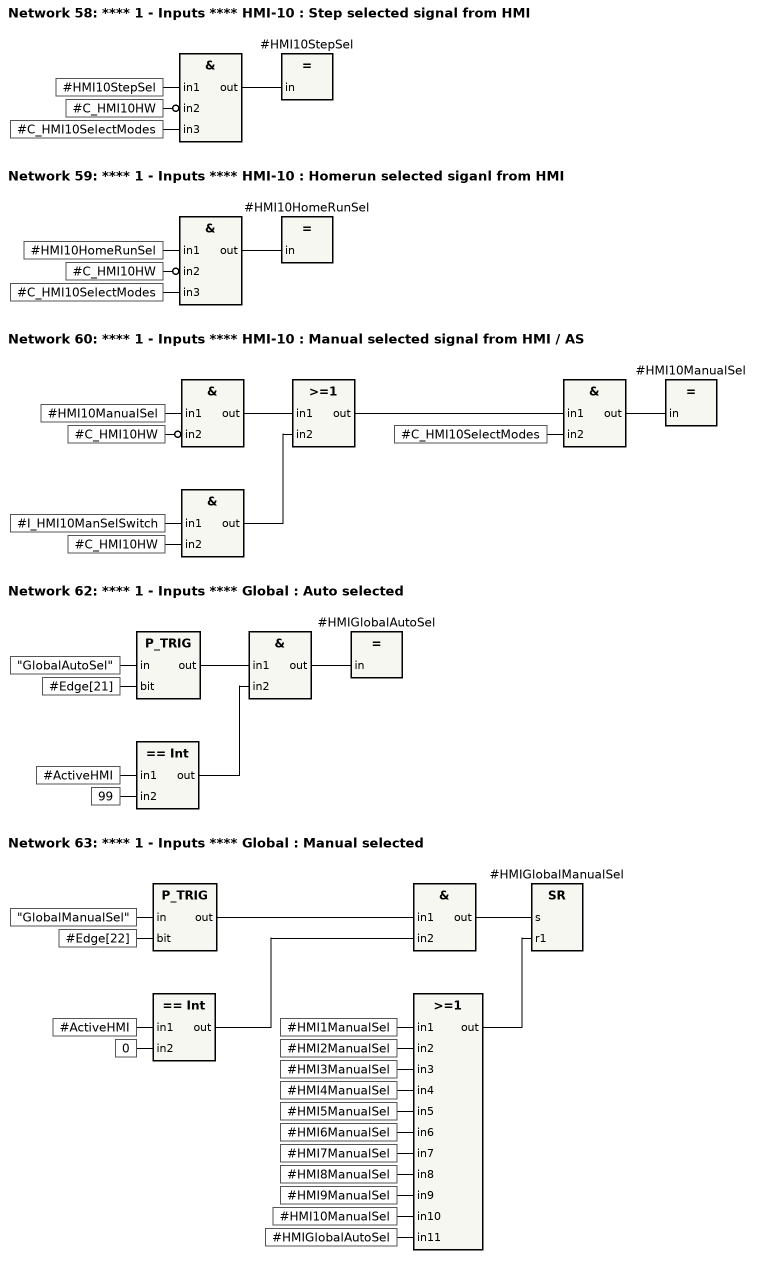
   #HMI10StepSel := #HMI10StepSel AND NOT #C_HMI10HW AND #C_HMI10SelectModes;
END_REGION

REGION Network 59: **** 1 - Inputs **** HMI-10 : Homerun selected siganl from HMI
   #HMI10HomeRunSel := #HMI10HomeRunSel AND NOT #C_HMI10HW AND #C_HMI10SelectModes;
END_REGION

REGION Network 60: **** 1 - Inputs **** HMI-10 : Manual selected signal from HMI / AS
   #HMI10ManualSel := ((#HMI10ManualSel AND NOT #C_HMI10HW) OR (#I_HMI10ManSelSwitch AND #C_HMI10HW)) AND #C_HMI10SelectModes;
END_REGION

REGION Network 61: ---------------------------------------------------------- Global ----------------------------------------------------------
END_REGION

REGION Network 62: **** 1 - Inputs **** Global : Auto selected
   #_w1 := "GlobalAutoSel" AND NOT #Edge[21];   // rising edge
   #Edge[21] := "GlobalAutoSel";
   #HMIGlobalAutoSel := #_w1 AND (#ActiveHMI = 99);
END_REGION

REGION Network 63: **** 1 - Inputs **** Global : Manual selected
   #_w1 := "GlobalManualSel" AND NOT #Edge[22];   // rising edge
   #Edge[22] := "GlobalManualSel";
   IF #_w1 AND (#ActiveHMI = 0) THEN
       #HMIGlobalManualSel := TRUE;   // SR flip-flop
   END_IF;
   IF #HMI1ManualSel OR #HMI2ManualSel OR #HMI3ManualSel OR #HMI4ManualSel OR #HMI5ManualSel OR #HMI6ManualSel OR #HMI7ManualSel OR #HMI8ManualSel OR #HMI9ManualSel OR #HMI10ManualSel OR #HMIGlobalAutoSel THEN
       #HMIGlobalManualSel := FALSE;
   END_IF;
END_REGION

REGION Network 64: ----------------------------------------------------------------------------------------------------------------------------------------------------------------------------
END_REGION

REGION Network 65: **** 1 - Inputs **** Extract the homerun modeselection from HMI
   // Extract the homerun modeselection from HMI
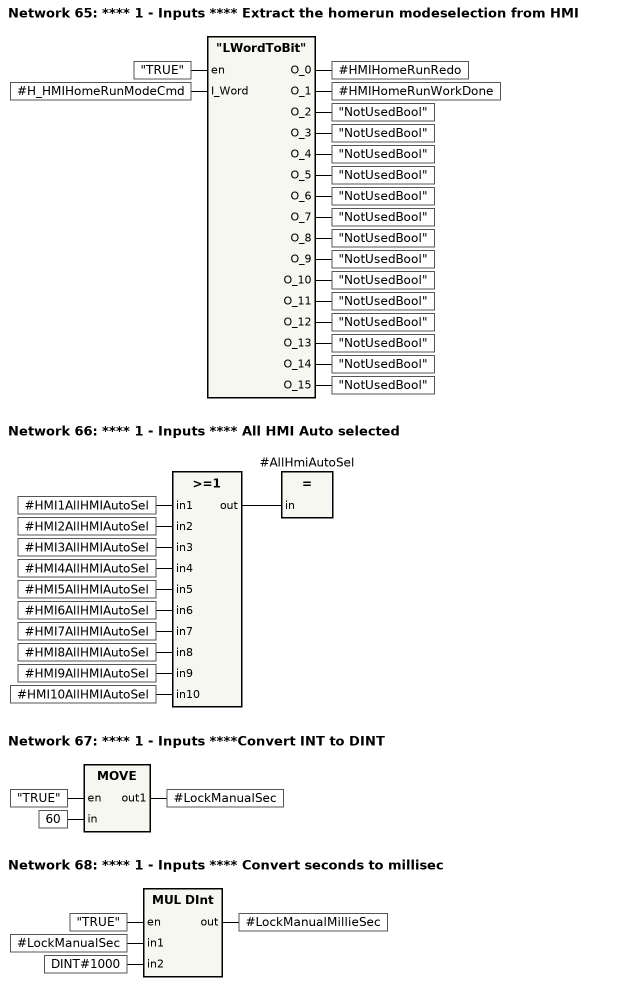
   IF "TRUE" THEN
       "LWordToBit"(I_Word := #H_HMIHomeRunModeCmd,
                    O_0 => #HMIHomeRunRedo,
                    O_1 => #HMIHomeRunWorkDone,
                    O_2 => "NotUsedBool",
                    O_3 => "NotUsedBool",
                    O_4 => "NotUsedBool",
                    O_5 => "NotUsedBool",
                    O_6 => "NotUsedBool",
                    O_7 => "NotUsedBool",
                    O_8 => "NotUsedBool",
                    O_9 => "NotUsedBool",
                    O_10 => "NotUsedBool",
                    O_11 => "NotUsedBool",
                    O_12 => "NotUsedBool",
                    O_13 => "NotUsedBool",
                    O_14 => "NotUsedBool",
                    O_15 => "NotUsedBool");
   END_IF;
END_REGION

REGION Network 66: **** 1 - Inputs **** All HMI Auto selected
   // All HMI Auto selected
   #AllHmiAutoSel := #HMI1AllHMIAutoSel OR #HMI2AllHMIAutoSel OR #HMI3AllHMIAutoSel OR #HMI4AllHMIAutoSel OR #HMI5AllHMIAutoSel OR #HMI6AllHMIAutoSel OR #HMI7AllHMIAutoSel OR #HMI8AllHMIAutoSel OR #HMI9AllHMIAutoSel OR #HMI10AllHMIAutoSel;
END_REGION

REGION Network 67: **** 1 - Inputs ****Convert INT to DINT
   // Convert INT to DINT
   IF "TRUE" THEN #LockManualSec := 60; END_IF;
END_REGION

REGION Network 68: **** 1 - Inputs **** Convert seconds to millisec
   // Convert seconds to millisec
   IF "TRUE" THEN #LockManualMillieSec := #LockManualSec * DINT#1000; END_IF;
END_REGION

REGION Network 69: **** 1 - Inputs **** Summary of all start buttons
   // Summary of all start buttons
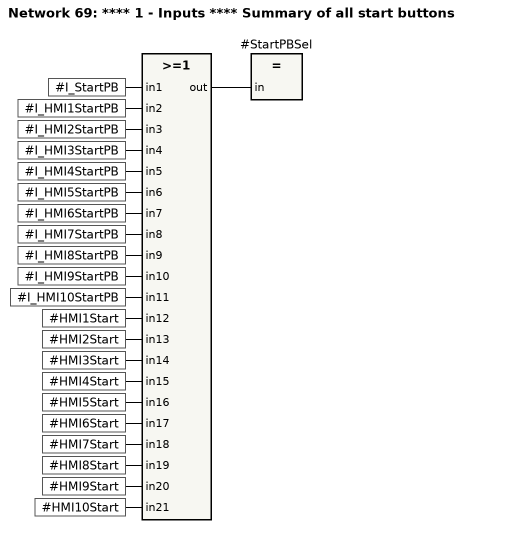
   #StartPBSel := #I_StartPB OR #I_HMI1StartPB OR #I_HMI2StartPB OR #I_HMI3StartPB OR #I_HMI4StartPB OR #I_HMI5StartPB OR #I_HMI6StartPB OR #I_HMI7StartPB OR #I_HMI8StartPB OR #I_HMI9StartPB OR #I_HMI10StartPB OR #HMI1Start OR #HMI2Start OR #HMI3Start OR #HMI4Start OR #HMI5Start OR #HMI6Start OR #HMI7Start OR #HMI8Start OR #HMI9Start OR #HMI10Start;
END_REGION

REGION Network 70: **** 1 - Inputs **** Reset Start button from HMI
   // Reset Start button from HMI
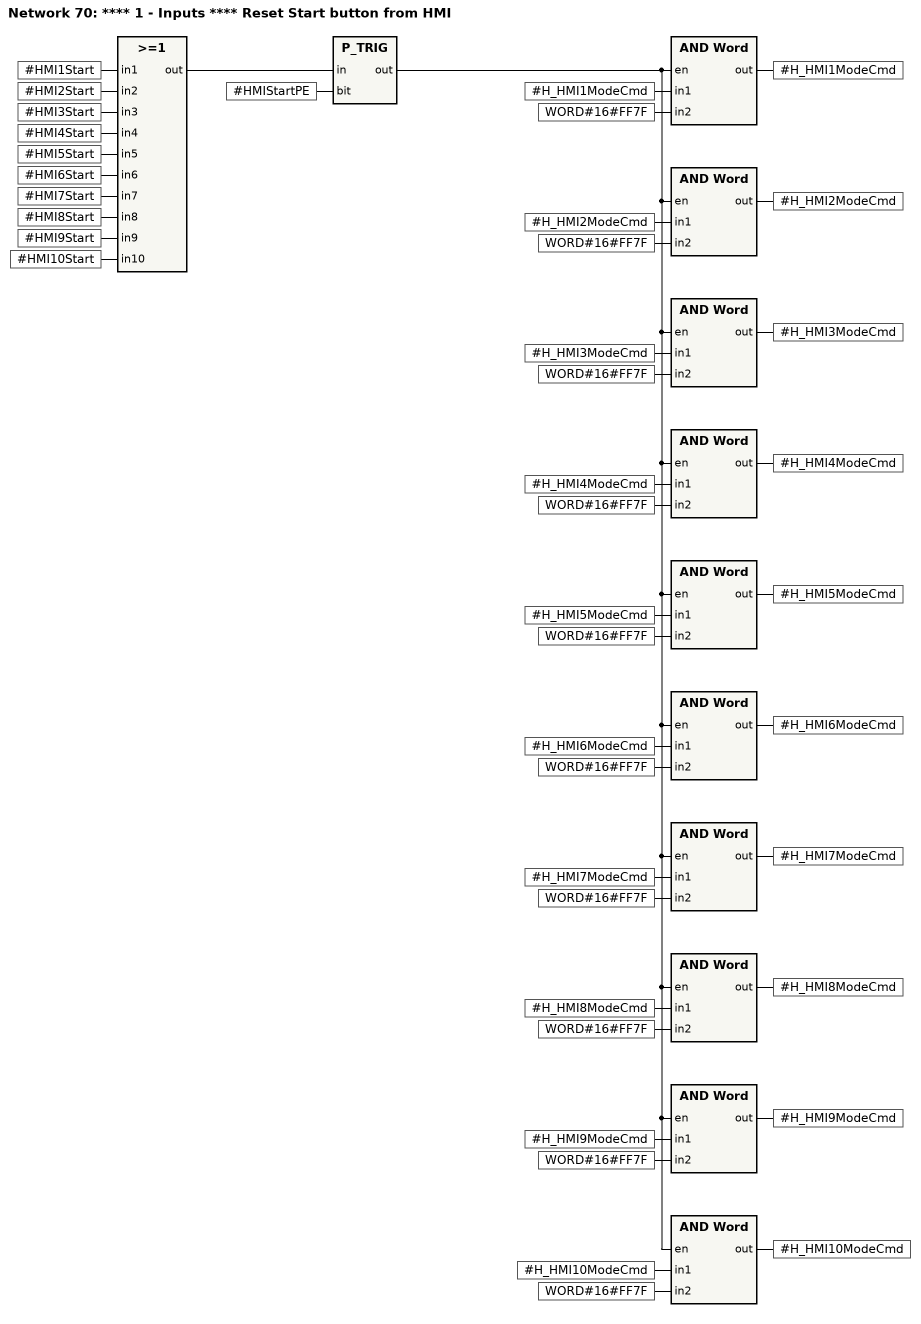
   #_w1 := #HMI1Start OR #HMI2Start OR #HMI3Start OR #HMI4Start OR #HMI5Start OR #HMI6Start OR #HMI7Start OR #HMI8Start OR #HMI9Start OR #HMI10Start;
   #_w2 := #_w1 AND NOT #HMIStartPE;   // rising edge
   #HMIStartPE := #_w1;
   IF #_w2 THEN
       #H_HMI1ModeCmd := #H_HMI1ModeCmd AND WORD#16#FF7F;
       #H_HMI2ModeCmd := #H_HMI2ModeCmd AND WORD#16#FF7F;
       #H_HMI3ModeCmd := #H_HMI3ModeCmd AND WORD#16#FF7F;
       #H_HMI4ModeCmd := #H_HMI4ModeCmd AND WORD#16#FF7F;
       #H_HMI5ModeCmd := #H_HMI5ModeCmd AND WORD#16#FF7F;
       #H_HMI6ModeCmd := #H_HMI6ModeCmd AND WORD#16#FF7F;
       #H_HMI7ModeCmd := #H_HMI7ModeCmd AND WORD#16#FF7F;
       #H_HMI8ModeCmd := #H_HMI8ModeCmd AND WORD#16#FF7F;
       #H_HMI9ModeCmd := #H_HMI9ModeCmd AND WORD#16#FF7F;
       #H_HMI10ModeCmd := #H_HMI10ModeCmd AND WORD#16#FF7F;
   END_IF;
END_REGION

REGION Network 71: **** 1 - Inputs **** Summary of all alarm reset buttons
   // Summary of all alarm reset buttons
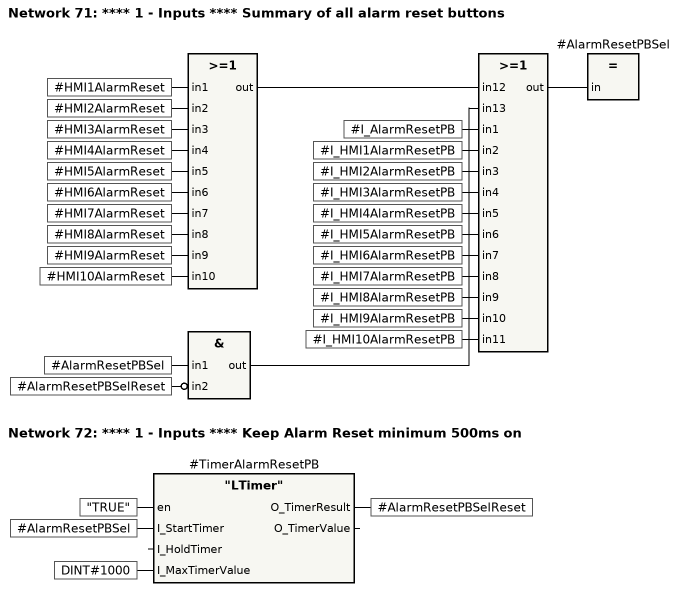
   #AlarmResetPBSel := #HMI1AlarmReset OR #HMI2AlarmReset OR #HMI3AlarmReset OR #HMI4AlarmReset OR #HMI5AlarmReset OR #HMI6AlarmReset OR #HMI7AlarmReset OR #HMI8AlarmReset OR #HMI9AlarmReset OR #HMI10AlarmReset OR (#AlarmResetPBSel AND NOT #AlarmResetPBSelReset) OR #I_AlarmResetPB OR #I_HMI1AlarmResetPB OR #I_HMI2AlarmResetPB OR #I_HMI3AlarmResetPB OR #I_HMI4AlarmResetPB OR #I_HMI5AlarmResetPB OR #I_HMI6AlarmResetPB OR #I_HMI7AlarmResetPB OR #I_HMI8AlarmResetPB OR #I_HMI9AlarmResetPB OR #I_HMI10AlarmResetPB;
END_REGION

REGION Network 72: **** 1 - Inputs **** Keep Alarm Reset minimum 500ms on
   // Keep Alarm Reset minimum 500ms on
   IF "TRUE" THEN
       #TimerAlarmResetPB(I_StartTimer := #AlarmResetPBSel,   // "LTimer"
                          I_MaxTimerValue := DINT#1000,
                          O_TimerResult => #AlarmResetPBSelReset);
   END_IF;
END_REGION

REGION Network 73: **** 1 - Inputs **** Reset AlarmResetPb from HMI
   // Reset AlarmResetPb from HMI
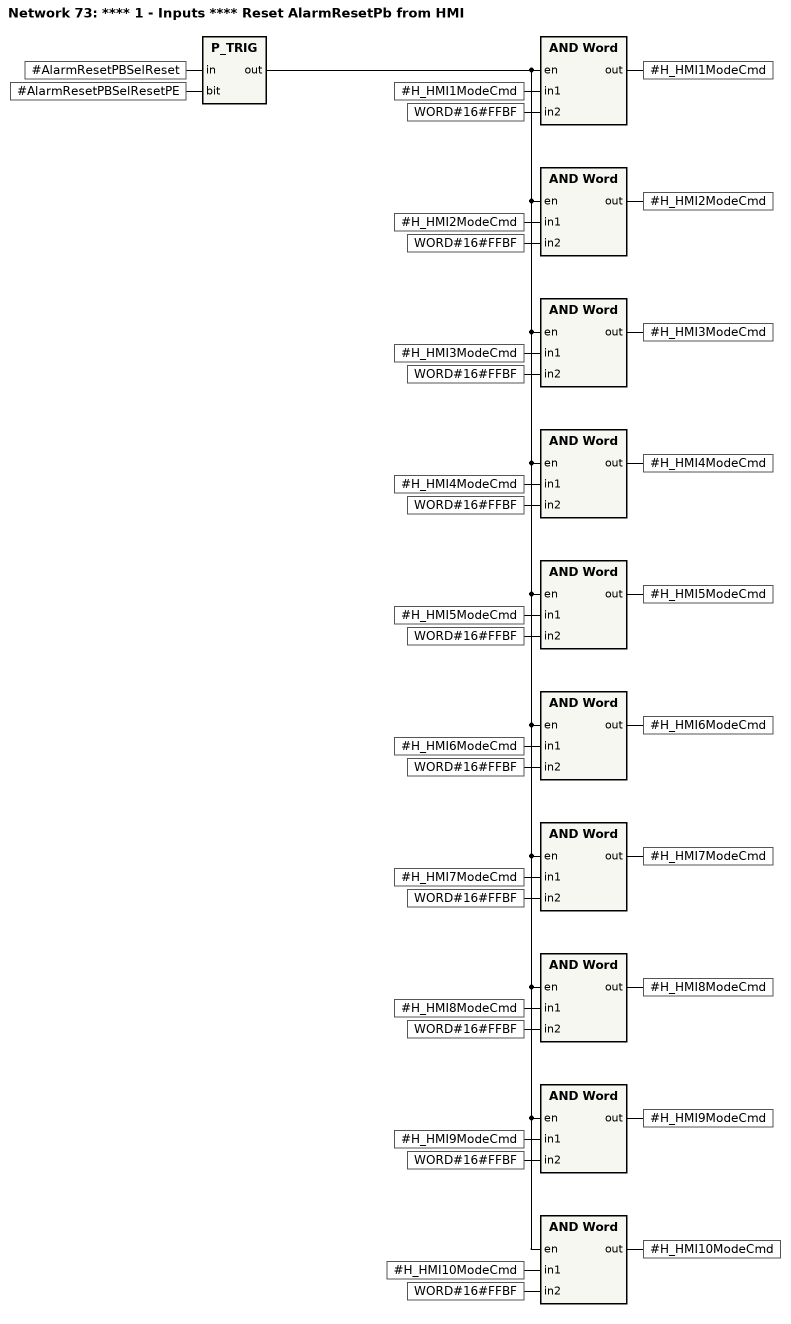
   #_w1 := #AlarmResetPBSelReset AND NOT #AlarmResetPBSelResetPE;   // rising edge
   #AlarmResetPBSelResetPE := #AlarmResetPBSelReset;
   IF #_w1 THEN
       #H_HMI1ModeCmd := #H_HMI1ModeCmd AND WORD#16#FFBF;
       #H_HMI2ModeCmd := #H_HMI2ModeCmd AND WORD#16#FFBF;
       #H_HMI3ModeCmd := #H_HMI3ModeCmd AND WORD#16#FFBF;
       #H_HMI4ModeCmd := #H_HMI4ModeCmd AND WORD#16#FFBF;
       #H_HMI5ModeCmd := #H_HMI5ModeCmd AND WORD#16#FFBF;
       #H_HMI6ModeCmd := #H_HMI6ModeCmd AND WORD#16#FFBF;
       #H_HMI7ModeCmd := #H_HMI7ModeCmd AND WORD#16#FFBF;
       #H_HMI8ModeCmd := #H_HMI8ModeCmd AND WORD#16#FFBF;
       #H_HMI9ModeCmd := #H_HMI9ModeCmd AND WORD#16#FFBF;
       #H_HMI10ModeCmd := #H_HMI10ModeCmd AND WORD#16#FFBF;
   END_IF;
END_REGION

REGION Network 74: **** 1 - Inputs **** Reset AlarmResetAckPb from HMI
   // Reset AlarmResetAckPb from HMI
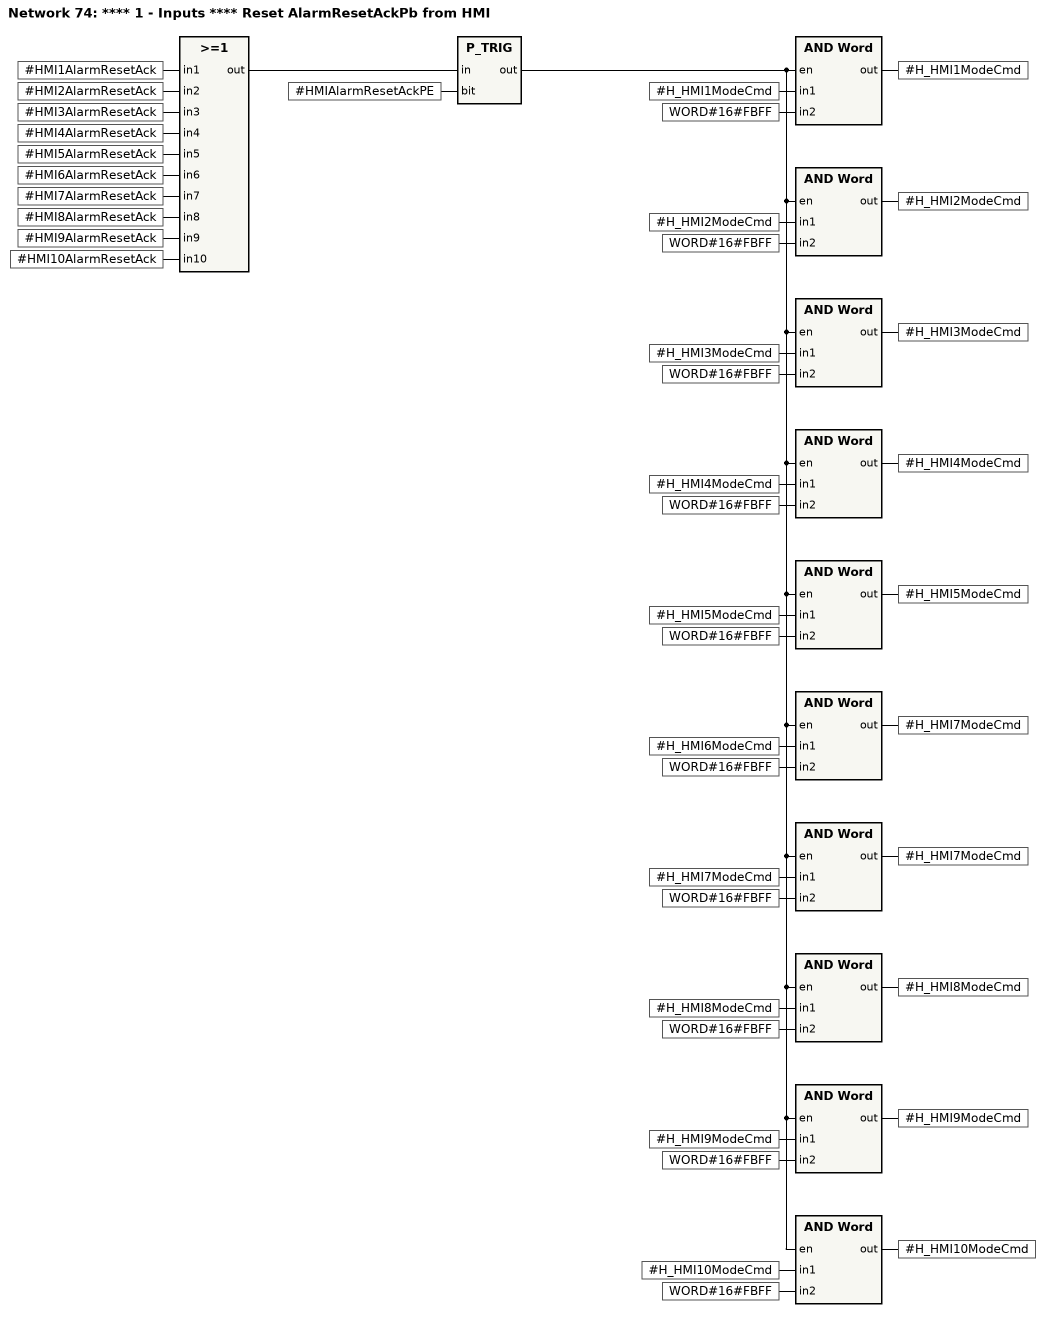
   #_w1 := #HMI1AlarmResetAck OR #HMI2AlarmResetAck OR #HMI3AlarmResetAck OR #HMI4AlarmResetAck OR #HMI5AlarmResetAck OR #HMI6AlarmResetAck OR #HMI7AlarmResetAck OR #HMI8AlarmResetAck OR #HMI9AlarmResetAck OR #HMI10AlarmResetAck;
   #_w2 := #_w1 AND NOT #HMIAlarmResetAckPE;   // rising edge
   #HMIAlarmResetAckPE := #_w1;
   IF #_w2 THEN
       #H_HMI1ModeCmd := #H_HMI1ModeCmd AND WORD#16#FBFF;
       #H_HMI2ModeCmd := #H_HMI2ModeCmd AND WORD#16#FBFF;
       #H_HMI3ModeCmd := #H_HMI3ModeCmd AND WORD#16#FBFF;
       #H_HMI4ModeCmd := #H_HMI4ModeCmd AND WORD#16#FBFF;
       #H_HMI5ModeCmd := #H_HMI5ModeCmd AND WORD#16#FBFF;
       #H_HMI7ModeCmd := #H_HMI6ModeCmd AND WORD#16#FBFF;
       #H_HMI7ModeCmd := #H_HMI7ModeCmd AND WORD#16#FBFF;
       #H_HMI8ModeCmd := #H_HMI8ModeCmd AND WORD#16#FBFF;
       #H_HMI9ModeCmd := #H_HMI9ModeCmd AND WORD#16#FBFF;
       #H_HMI10ModeCmd := #H_HMI10ModeCmd AND WORD#16#FBFF;
   END_IF;
END_REGION

REGION Network 75: **** 1 - Inputs **** Reset ResetTM button from HMI
   // Reset ResetTM button from HMI
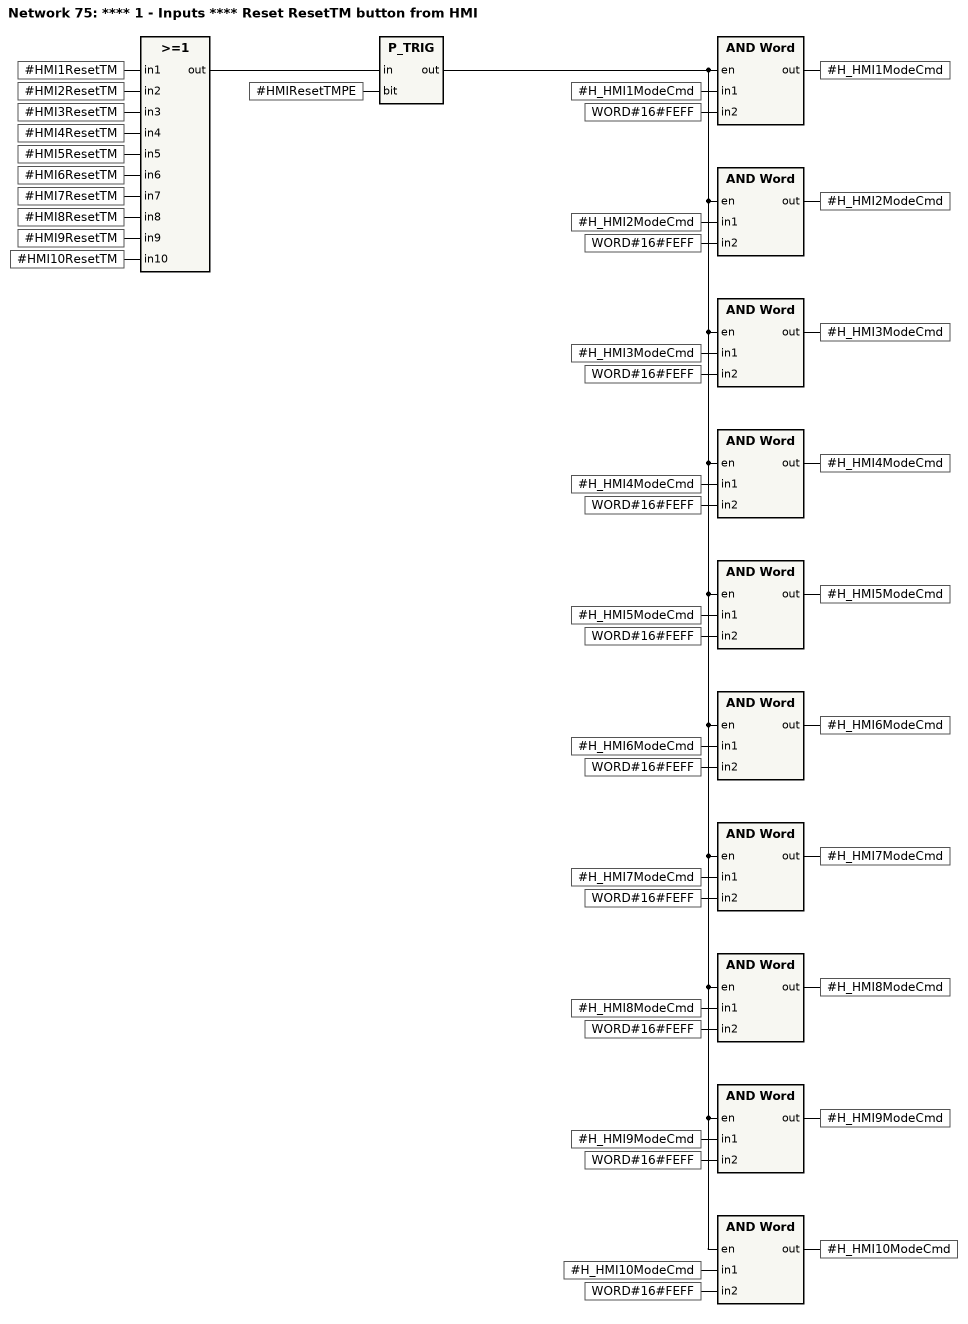
   #_w1 := #HMI1ResetTM OR #HMI2ResetTM OR #HMI3ResetTM OR #HMI4ResetTM OR #HMI5ResetTM OR #HMI6ResetTM OR #HMI7ResetTM OR #HMI8ResetTM OR #HMI9ResetTM OR #HMI10ResetTM;
   #_w2 := #_w1 AND NOT #HMIResetTMPE;   // rising edge
   #HMIResetTMPE := #_w1;
   IF #_w2 THEN
       #H_HMI1ModeCmd := #H_HMI1ModeCmd AND WORD#16#FEFF;
       #H_HMI2ModeCmd := #H_HMI2ModeCmd AND WORD#16#FEFF;
       #H_HMI3ModeCmd := #H_HMI3ModeCmd AND WORD#16#FEFF;
       #H_HMI4ModeCmd := #H_HMI4ModeCmd AND WORD#16#FEFF;
       #H_HMI5ModeCmd := #H_HMI5ModeCmd AND WORD#16#FEFF;
       #H_HMI6ModeCmd := #H_HMI6ModeCmd AND WORD#16#FEFF;
       #H_HMI7ModeCmd := #H_HMI7ModeCmd AND WORD#16#FEFF;
       #H_HMI8ModeCmd := #H_HMI8ModeCmd AND WORD#16#FEFF;
       #H_HMI9ModeCmd := #H_HMI9ModeCmd AND WORD#16#FEFF;
       #H_HMI10ModeCmd := #H_HMI10ModeCmd AND WORD#16#FEFF;
   END_IF;
END_REGION

REGION Network 76: **** 1 - Inputs **** Reset ResetSeq button from HMI
   // Reset ResetSeq button from HMI
